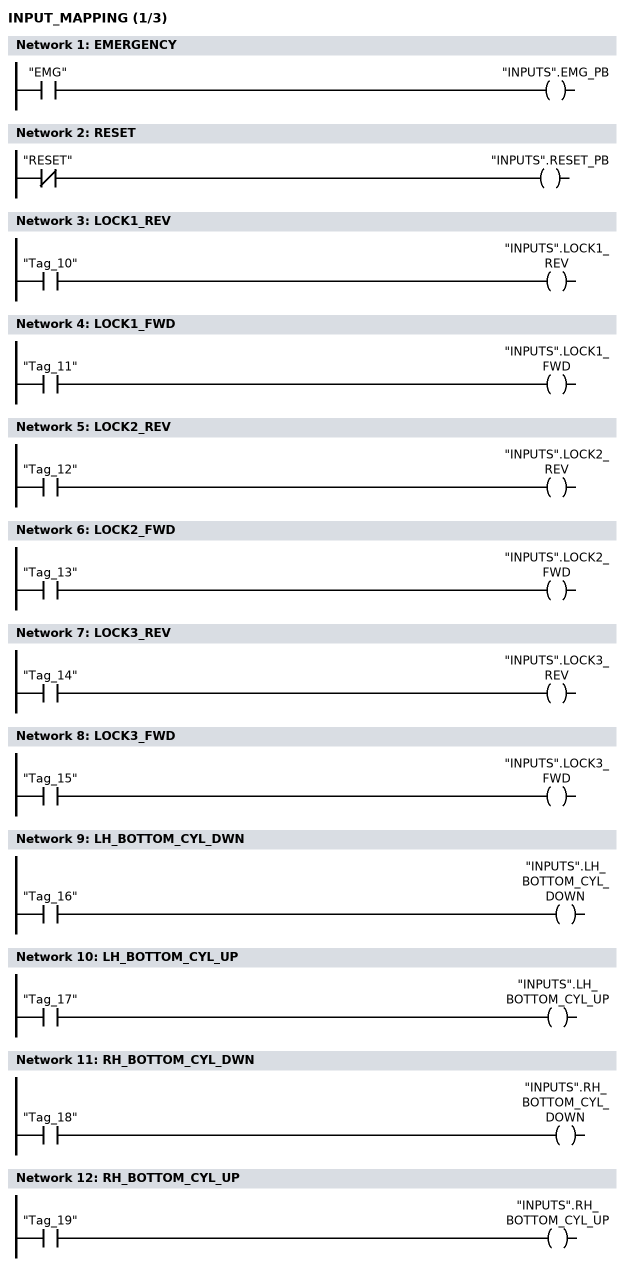
   RUNG wire#powerrail
      Contact( "EMG" )
      Coil( "INPUTS".EMG_PB )
   END_RUNG
   // the same network as SCL:
   "INPUTS".EMG_PB := "EMG";
END_REGION

REGION Network 2: RESET
   RUNG wire#powerrail
      I_Contact( "RESET" )
      Coil( "INPUTS".RESET_PB )
   END_RUNG
   // the same network as SCL:
   "INPUTS".RESET_PB := NOT "RESET";
END_REGION

REGION Network 3: LOCK1_REV
   RUNG wire#powerrail
      Contact( "Tag_10" )
      Coil( "INPUTS".LOCK1_REV )
   END_RUNG
   // the same network as SCL:
   "INPUTS".LOCK1_REV := "Tag_10";
END_REGION

REGION Network 4: LOCK1_FWD
   RUNG wire#powerrail
      Contact( "Tag_11" )
      Coil( "INPUTS".LOCK1_FWD )
   END_RUNG
   // the same network as SCL:
   "INPUTS".LOCK1_FWD := "Tag_11";
END_REGION

REGION Network 5: LOCK2_REV
   RUNG wire#powerrail
      Contact( "Tag_12" )
      Coil( "INPUTS".LOCK2_REV )
   END_RUNG
   // the same network as SCL:
   "INPUTS".LOCK2_REV := "Tag_12";
END_REGION

REGION Network 6: LOCK2_FWD
   RUNG wire#powerrail
      Contact( "Tag_13" )
      Coil( "INPUTS".LOCK2_FWD )
   END_RUNG
   // the same network as SCL:
   "INPUTS".LOCK2_FWD := "Tag_13";
END_REGION

REGION Network 7: LOCK3_REV
   RUNG wire#powerrail
      Contact( "Tag_14" )
      Coil( "INPUTS".LOCK3_REV )
   END_RUNG
   // the same network as SCL:
   "INPUTS".LOCK3_REV := "Tag_14";
END_REGION

REGION Network 8: LOCK3_FWD
   RUNG wire#powerrail
      Contact( "Tag_15" )
      Coil( "INPUTS".LOCK3_FWD )
   END_RUNG
   // the same network as SCL:
   "INPUTS".LOCK3_FWD := "Tag_15";
END_REGION

REGION Network 9: LH_BOTTOM_CYL_DWN
   RUNG wire#powerrail
      Contact( "Tag_16" )
      Coil( "INPUTS".LH_BOTTOM_CYL_DOWN )
   END_RUNG
   // the same network as SCL:
   "INPUTS".LH_BOTTOM_CYL_DOWN := "Tag_16";
END_REGION

REGION Network 10: LH_BOTTOM_CYL_UP
   RUNG wire#powerrail
      Contact( "Tag_17" )
      Coil( "INPUTS".LH_BOTTOM_CYL_UP )
   END_RUNG
   // the same network as SCL:
   "INPUTS".LH_BOTTOM_CYL_UP := "Tag_17";
END_REGION

REGION Network 11: RH_BOTTOM_CYL_DWN
   RUNG wire#powerrail
      Contact( "Tag_18" )
      Coil( "INPUTS".RH_BOTTOM_CYL_DOWN )
   END_RUNG
   // the same network as SCL:
   "INPUTS".RH_BOTTOM_CYL_DOWN := "Tag_18";
END_REGION

REGION Network 12: RH_BOTTOM_CYL_UP
   RUNG wire#powerrail
      Contact( "Tag_19" )
      Coil( "INPUTS".RH_BOTTOM_CYL_UP )
   END_RUNG
   // the same network as SCL:
   "INPUTS".RH_BOTTOM_CYL_UP := "Tag_19";
END_REGION

REGION Network 13: PUNCH_CYL1_REV
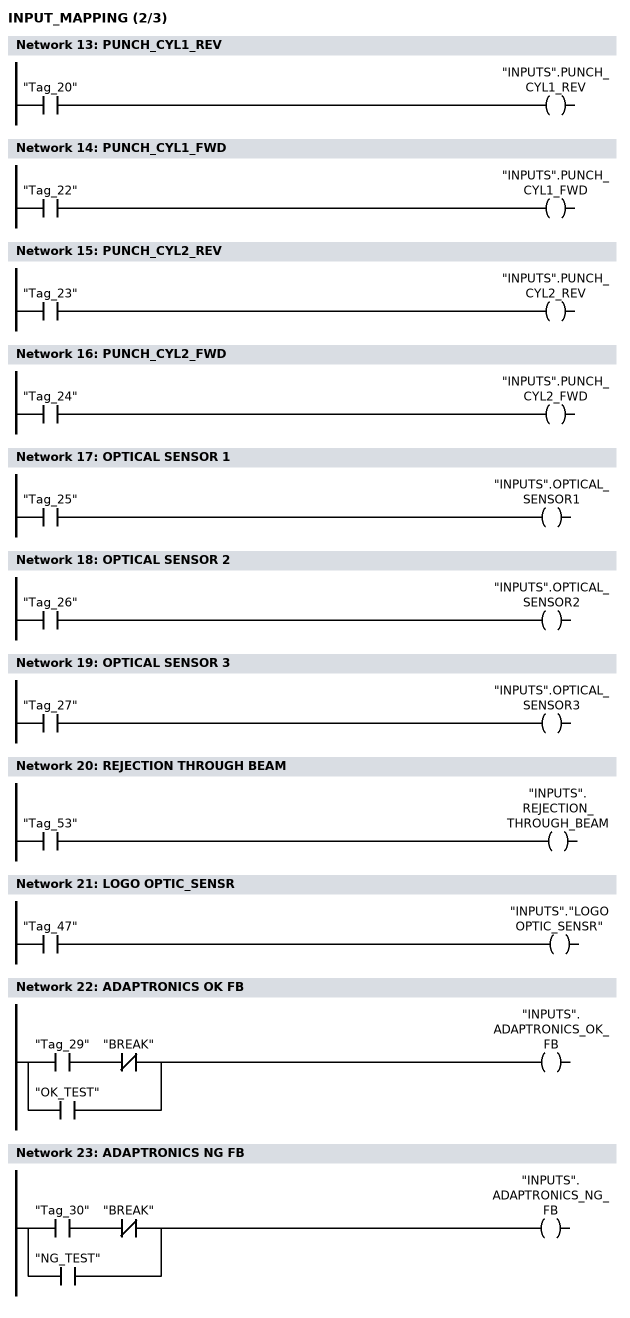
   RUNG wire#powerrail
      Contact( "Tag_20" )
      Coil( "INPUTS".PUNCH_CYL1_REV )
   END_RUNG
   // the same network as SCL:
   "INPUTS".PUNCH_CYL1_REV := "Tag_20";
END_REGION

REGION Network 14: PUNCH_CYL1_FWD
   RUNG wire#powerrail
      Contact( "Tag_22" )
      Coil( "INPUTS".PUNCH_CYL1_FWD )
   END_RUNG
   // the same network as SCL:
   "INPUTS".PUNCH_CYL1_FWD := "Tag_22";
END_REGION

REGION Network 15: PUNCH_CYL2_REV
   RUNG wire#powerrail
      Contact( "Tag_23" )
      Coil( "INPUTS".PUNCH_CYL2_REV )
   END_RUNG
   // the same network as SCL:
   "INPUTS".PUNCH_CYL2_REV := "Tag_23";
END_REGION

REGION Network 16: PUNCH_CYL2_FWD
   RUNG wire#powerrail
      Contact( "Tag_24" )
      Coil( "INPUTS".PUNCH_CYL2_FWD )
   END_RUNG
   // the same network as SCL:
   "INPUTS".PUNCH_CYL2_FWD := "Tag_24";
END_REGION

REGION Network 17: OPTICAL SENSOR 1
   RUNG wire#powerrail
      Contact( "Tag_25" )
      Coil( "INPUTS".OPTICAL_SENSOR1 )
   END_RUNG
   // the same network as SCL:
   "INPUTS".OPTICAL_SENSOR1 := "Tag_25";
END_REGION

REGION Network 18: OPTICAL SENSOR 2
   RUNG wire#powerrail
      Contact( "Tag_26" )
      Coil( "INPUTS".OPTICAL_SENSOR2 )
   END_RUNG
   // the same network as SCL:
   "INPUTS".OPTICAL_SENSOR2 := "Tag_26";
END_REGION

REGION Network 19: OPTICAL SENSOR 3
   RUNG wire#powerrail
      Contact( "Tag_27" )
      Coil( "INPUTS".OPTICAL_SENSOR3 )
   END_RUNG
   // the same network as SCL:
   "INPUTS".OPTICAL_SENSOR3 := "Tag_27";
END_REGION

REGION Network 20: REJECTION THROUGH BEAM
   RUNG wire#powerrail
      Contact( "Tag_53" )
      Coil( "INPUTS".REJECTION_THROUGH_BEAM )
   END_RUNG
   // the same network as SCL:
   "INPUTS".REJECTION_THROUGH_BEAM := "Tag_53";
END_REGION

REGION Network 21: LOGO OPTIC_SENSR
   RUNG wire#powerrail
      Contact( "Tag_47" )
      Coil( "INPUTS"."LOGO OPTIC_SENSR" )
   END_RUNG
   // the same network as SCL:
   "INPUTS"."LOGO OPTIC_SENSR" := "Tag_47";
END_REGION

REGION Network 22: ADAPTRONICS OK FB
   RUNG wire#powerrail
      Contact( "Tag_29" )
      I_Contact( "BREAK" )
      wire#w1
      Coil( "INPUTS".ADAPTRONICS_OK_FB )
   END_RUNG
   RUNG wire#powerrail
      Contact( "OK_TEST" )
   END_RUNG wire#w1
   // the same network as SCL:
   "INPUTS".ADAPTRONICS_OK_FB := ("Tag_29" AND NOT "BREAK") OR "OK_TEST";
END_REGION

REGION Network 23: ADAPTRONICS NG FB
   RUNG wire#powerrail
      Contact( "Tag_30" )
      I_Contact( "BREAK" )
      wire#w1
      Coil( "INPUTS".ADAPTRONICS_NG_FB )
   END_RUNG
   RUNG wire#powerrail
      Contact( "NG_TEST" )
   END_RUNG wire#w1
   // the same network as SCL:
   "INPUTS".ADAPTRONICS_NG_FB := ("Tag_30" AND NOT "BREAK") OR "NG_TEST";
END_REGION

REGION Network 24: ADAPTRONICS SEGMENT FB
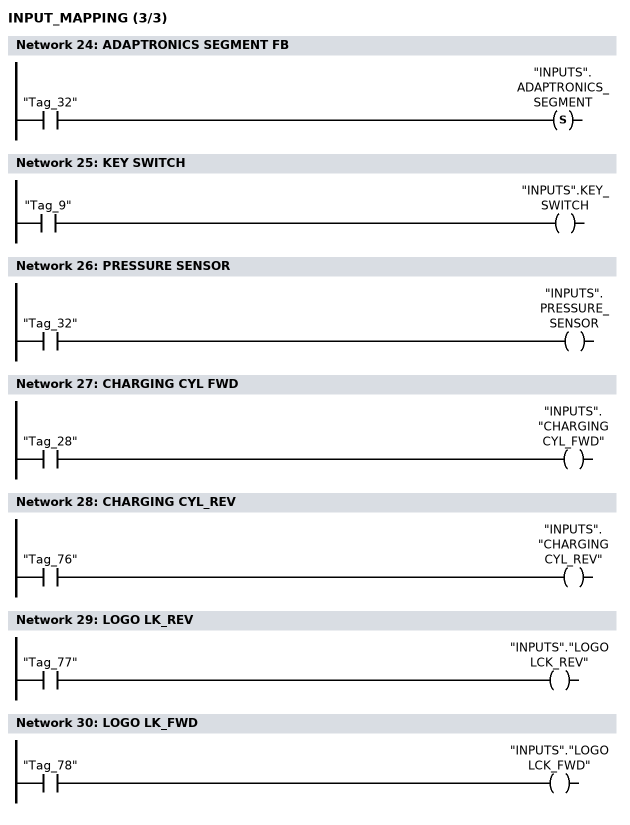
   RUNG wire#powerrail
      Contact( "Tag_32" )
      S_Coil( "INPUTS".ADAPTRONICS_SEGMENT )
   END_RUNG
   // the same network as SCL:
   IF "Tag_32" THEN "INPUTS".ADAPTRONICS_SEGMENT := TRUE; END_IF;
END_REGION

REGION Network 25: KEY SWITCH
   RUNG wire#powerrail
      Contact( "Tag_9" )
      Coil( "INPUTS".KEY_SWITCH )
   END_RUNG
   // the same network as SCL:
   "INPUTS".KEY_SWITCH := "Tag_9";
END_REGION

REGION Network 26: PRESSURE SENSOR
   RUNG wire#powerrail
      Contact( "Tag_32" )
      Coil( "INPUTS".PRESSURE_SENSOR )
   END_RUNG
   // the same network as SCL:
   "INPUTS".PRESSURE_SENSOR := "Tag_32";
END_REGION

REGION Network 27: CHARGING CYL FWD
   RUNG wire#powerrail
      Contact( "Tag_28" )
      Coil( "INPUTS"."CHARGING CYL_FWD" )
   END_RUNG
   // the same network as SCL:
   "INPUTS"."CHARGING CYL_FWD" := "Tag_28";
END_REGION

REGION Network 28: CHARGING CYL_REV
   RUNG wire#powerrail
      Contact( "Tag_76" )
      Coil( "INPUTS"."CHARGING CYL_REV" )
   END_RUNG
   // the same network as SCL:
   "INPUTS"."CHARGING CYL_REV" := "Tag_76";
END_REGION

REGION Network 29: LOGO LK_REV
   RUNG wire#powerrail
      Contact( "Tag_77" )
      Coil( "INPUTS"."LOGO LCK_REV" )
   END_RUNG
   // the same network as SCL:
   "INPUTS"."LOGO LCK_REV" := "Tag_77";
END_REGION

REGION Network 30: LOGO LK_FWD
   RUNG wire#powerrail
      Contact( "Tag_78" )
      Coil( "INPUTS"."LOGO LCK_FWD" )
   END_RUNG
   // the same network as SCL:
   "INPUTS"."LOGO LCK_FWD" := "Tag_78";
END_REGION
END_FUNCTION

FUNCTION "OUTPUT_MAPPING" : Void   // FC2, LAD
{ S7_Optimized_Access := 'TRUE' }
VERSION : 0.1
   VAR CONSTANT
      AMBER_ON : Bool;
   END_VAR
BEGIN

REGION Network 1: BUZZER
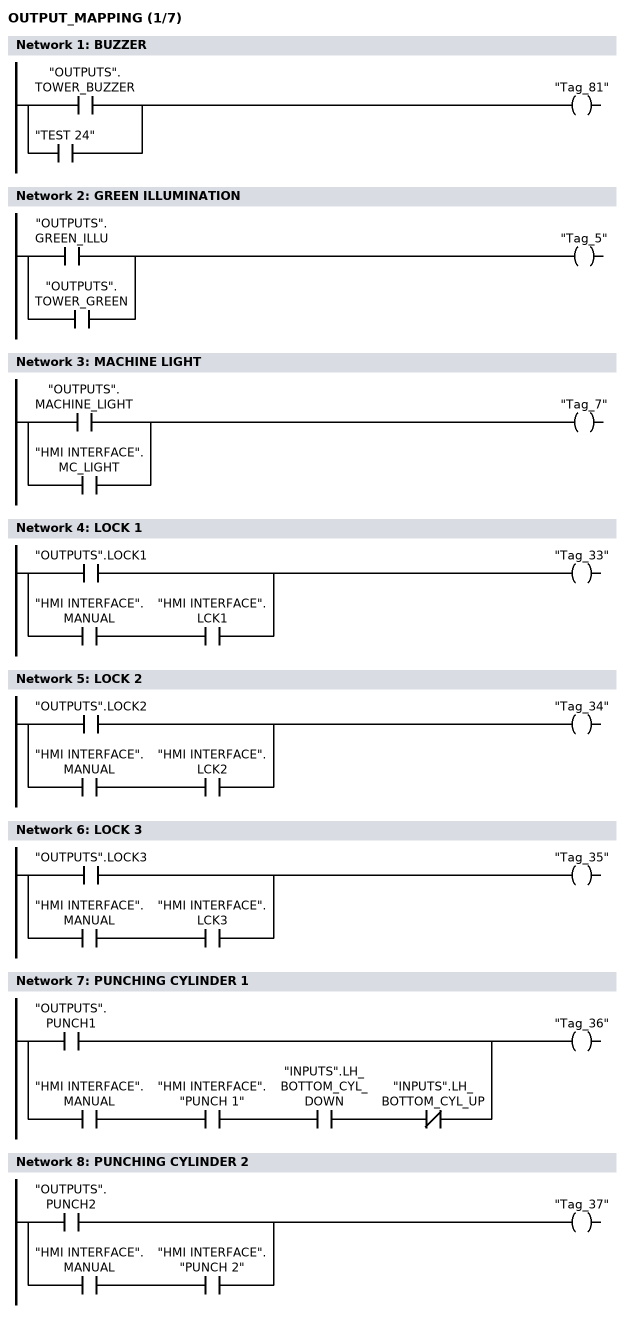
   RUNG wire#powerrail
      Contact( "OUTPUTS".TOWER_BUZZER )
      wire#w1
      Coil( "Tag_81" )
   END_RUNG
   RUNG wire#powerrail
      Contact( "TEST 24" )
   END_RUNG wire#w1
   // the same network as SCL:
   "Tag_81" := "OUTPUTS".TOWER_BUZZER OR "TEST 24";
END_REGION

REGION Network 2: GREEN ILLUMINATION
   RUNG wire#powerrail
      Contact( "OUTPUTS".GREEN_ILLU )
      wire#w1
      Coil( "Tag_5" )
   END_RUNG
   RUNG wire#powerrail
      Contact( "OUTPUTS".TOWER_GREEN )
   END_RUNG wire#w1
   // the same network as SCL:
   "Tag_5" := "OUTPUTS".GREEN_ILLU OR "OUTPUTS".TOWER_GREEN;
END_REGION

REGION Network 3: MACHINE LIGHT
   RUNG wire#powerrail
      Contact( "OUTPUTS".MACHINE_LIGHT )
      wire#w1
      Coil( "Tag_7" )
   END_RUNG
   RUNG wire#powerrail
      Contact( "HMI INTERFACE".MC_LIGHT )
   END_RUNG wire#w1
   // the same network as SCL:
   "Tag_7" := "OUTPUTS".MACHINE_LIGHT OR "HMI INTERFACE".MC_LIGHT;
END_REGION

REGION Network 4: LOCK 1
   RUNG wire#powerrail
      Contact( "OUTPUTS".LOCK1 )
      wire#w1
      Coil( "Tag_33" )
   END_RUNG
   RUNG wire#powerrail
      Contact( "HMI INTERFACE".MANUAL )
      Contact( "HMI INTERFACE".LCK1 )
   END_RUNG wire#w1
   // the same network as SCL:
   "Tag_33" := "OUTPUTS".LOCK1 OR ("HMI INTERFACE".MANUAL AND "HMI INTERFACE".LCK1);
END_REGION

REGION Network 5: LOCK 2
   RUNG wire#powerrail
      Contact( "OUTPUTS".LOCK2 )
      wire#w1
      Coil( "Tag_34" )
   END_RUNG
   RUNG wire#powerrail
      Contact( "HMI INTERFACE".MANUAL )
      Contact( "HMI INTERFACE".LCK2 )
   END_RUNG wire#w1
   // the same network as SCL:
   "Tag_34" := "OUTPUTS".LOCK2 OR ("HMI INTERFACE".MANUAL AND "HMI INTERFACE".LCK2);
END_REGION

REGION Network 6: LOCK 3
   RUNG wire#powerrail
      Contact( "OUTPUTS".LOCK3 )
      wire#w1
      Coil( "Tag_35" )
   END_RUNG
   RUNG wire#powerrail
      Contact( "HMI INTERFACE".MANUAL )
      Contact( "HMI INTERFACE".LCK3 )
   END_RUNG wire#w1
   // the same network as SCL:
   "Tag_35" := "OUTPUTS".LOCK3 OR ("HMI INTERFACE".MANUAL AND "HMI INTERFACE".LCK3);
END_REGION

REGION Network 7: PUNCHING CYLINDER 1
   RUNG wire#powerrail
      Contact( "OUTPUTS".PUNCH1 )
      wire#w1
      Coil( "Tag_36" )
   END_RUNG
   RUNG wire#powerrail
      Contact( "HMI INTERFACE".MANUAL )
      Contact( "HMI INTERFACE"."PUNCH 1" )
      Contact( "INPUTS".LH_BOTTOM_CYL_DOWN )
      I_Contact( "INPUTS".LH_BOTTOM_CYL_UP )
   END_RUNG wire#w1
   // the same network as SCL:
   "Tag_36" := "OUTPUTS".PUNCH1 OR ("HMI INTERFACE".MANUAL AND "HMI INTERFACE"."PUNCH 1" AND "INPUTS".LH_BOTTOM_CYL_DOWN AND NOT "INPUTS".LH_BOTTOM_CYL_UP);
END_REGION

REGION Network 8: PUNCHING CYLINDER 2
   RUNG wire#powerrail
      Contact( "OUTPUTS".PUNCH2 )
      wire#w1
      Coil( "Tag_37" )
   END_RUNG
   RUNG wire#powerrail
      Contact( "HMI INTERFACE".MANUAL )
      Contact( "HMI INTERFACE"."PUNCH 2" )
   END_RUNG wire#w1
   // the same network as SCL:
   "Tag_37" := "OUTPUTS".PUNCH2 OR ("HMI INTERFACE".MANUAL AND "HMI INTERFACE"."PUNCH 2");
END_REGION

REGION Network 9: LH_BOTTOM_CYL
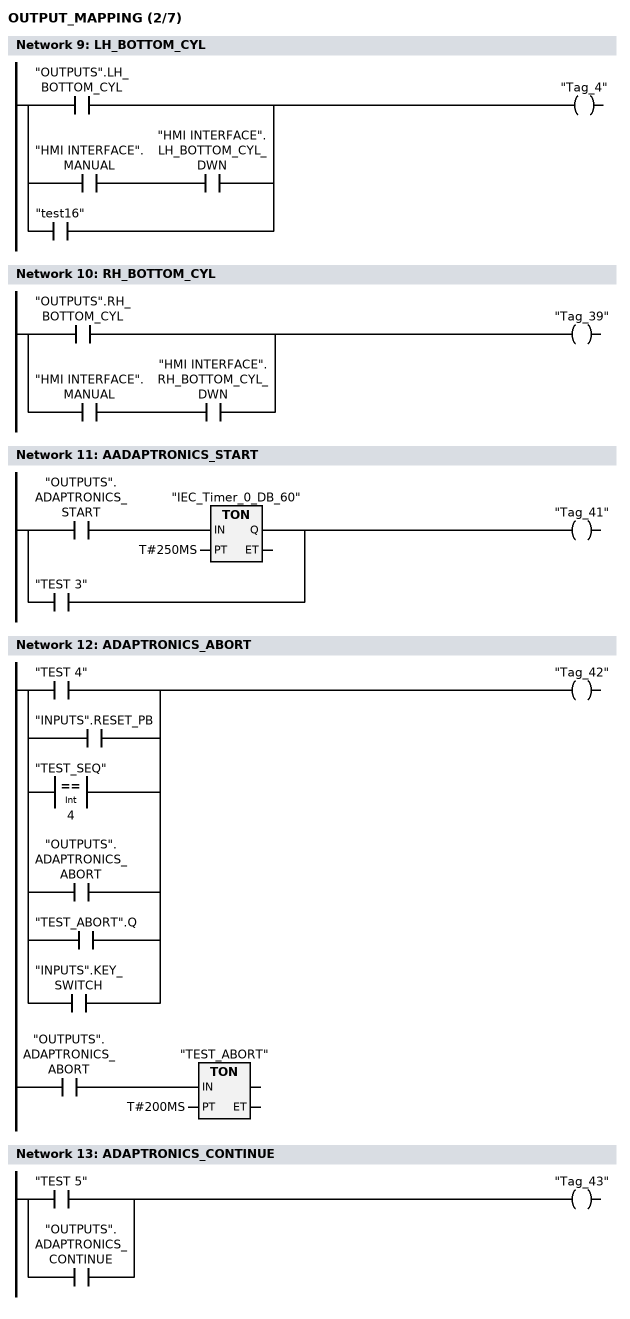
   RUNG wire#powerrail
      Contact( "OUTPUTS".LH_BOTTOM_CYL )
      wire#w1
      Coil( "Tag_4" )
   END_RUNG
   RUNG wire#powerrail
      Contact( "HMI INTERFACE".MANUAL )
      Contact( "HMI INTERFACE".LH_BOTTOM_CYL_DWN )
   END_RUNG wire#w1
   RUNG wire#powerrail
      Contact( "test16" )
   END_RUNG wire#w1
   // the same network as SCL:
   "Tag_4" := "OUTPUTS".LH_BOTTOM_CYL OR ("HMI INTERFACE".MANUAL AND "HMI INTERFACE".LH_BOTTOM_CYL_DWN) OR "test16";
END_REGION

REGION Network 10: RH_BOTTOM_CYL
   RUNG wire#powerrail
      Contact( "OUTPUTS".RH_BOTTOM_CYL )
      wire#w1
      Coil( "Tag_39" )
   END_RUNG
   RUNG wire#powerrail
      Contact( "HMI INTERFACE".MANUAL )
      Contact( "HMI INTERFACE".RH_BOTTOM_CYL_DWN )
   END_RUNG wire#w1
   // the same network as SCL:
   "Tag_39" := "OUTPUTS".RH_BOTTOM_CYL OR ("HMI INTERFACE".MANUAL AND "HMI INTERFACE".RH_BOTTOM_CYL_DWN);
END_REGION

REGION Network 11: AADAPTRONICS_START
   "IEC_Timer_0_DB_60".TON(IN := "OUTPUTS".ADAPTRONICS_START, PT := T#250MS);
   "Tag_41" := "IEC_Timer_0_DB_60".Q OR "TEST 3";
END_REGION

REGION Network 12: ADAPTRONICS_ABORT
   "Tag_42" := "TEST 4" OR "INPUTS".RESET_PB OR ("TEST_SEQ" = 4) OR "OUTPUTS".ADAPTRONICS_ABORT OR "TEST_ABORT".Q OR "INPUTS".KEY_SWITCH;
   "TEST_ABORT".TON(IN := "OUTPUTS".ADAPTRONICS_ABORT, PT := T#200MS);
END_REGION

REGION Network 13: ADAPTRONICS_CONTINUE
   RUNG wire#powerrail
      Contact( "TEST 5" )
      wire#w1
      Coil( "Tag_43" )
   END_RUNG
   RUNG wire#powerrail
      Contact( "OUTPUTS".ADAPTRONICS_CONTINUE )
   END_RUNG wire#w1
   // the same network as SCL:
   "Tag_43" := "TEST 5" OR "OUTPUTS".ADAPTRONICS_CONTINUE;
END_REGION

REGION Network 14: RELAY 1 / RED
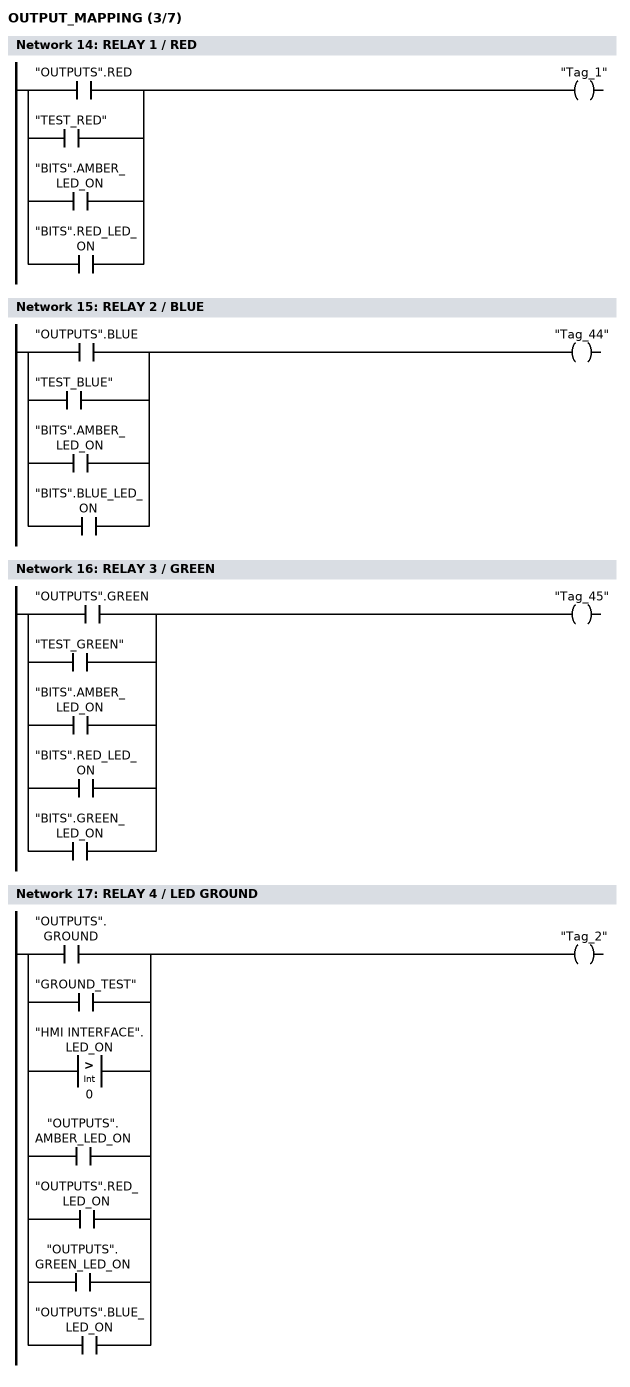
   RUNG wire#powerrail
      Contact( "OUTPUTS".RED )
      wire#w1
      Coil( "Tag_1" )
   END_RUNG
   RUNG wire#powerrail
      Contact( "TEST_RED" )
   END_RUNG wire#w1
   RUNG wire#powerrail
      Contact( "BITS".AMBER_LED_ON )
   END_RUNG wire#w1
   RUNG wire#powerrail
      Contact( "BITS".RED_LED_ON )
   END_RUNG wire#w1
   // the same network as SCL:
   "Tag_1" := "OUTPUTS".RED OR "TEST_RED" OR "BITS".AMBER_LED_ON OR "BITS".RED_LED_ON;
END_REGION

REGION Network 15: RELAY 2 / BLUE
   RUNG wire#powerrail
      Contact( "OUTPUTS".BLUE )
      wire#w1
      Coil( "Tag_44" )
   END_RUNG
   RUNG wire#powerrail
      Contact( "TEST_BLUE" )
   END_RUNG wire#w1
   RUNG wire#powerrail
      Contact( "BITS".AMBER_LED_ON )
   END_RUNG wire#w1
   RUNG wire#powerrail
      Contact( "BITS".BLUE_LED_ON )
   END_RUNG wire#w1
   // the same network as SCL:
   "Tag_44" := "OUTPUTS".BLUE OR "TEST_BLUE" OR "BITS".AMBER_LED_ON OR "BITS".BLUE_LED_ON;
END_REGION

REGION Network 16: RELAY 3 / GREEN
   RUNG wire#powerrail
      Contact( "OUTPUTS".GREEN )
      wire#w1
      Coil( "Tag_45" )
   END_RUNG
   RUNG wire#powerrail
      Contact( "TEST_GREEN" )
   END_RUNG wire#w1
   RUNG wire#powerrail
      Contact( "BITS".AMBER_LED_ON )
   END_RUNG wire#w1
   RUNG wire#powerrail
      Contact( "BITS".RED_LED_ON )
   END_RUNG wire#w1
   RUNG wire#powerrail
      Contact( "BITS".GREEN_LED_ON )
   END_RUNG wire#w1
   // the same network as SCL:
   "Tag_45" := "OUTPUTS".GREEN OR "TEST_GREEN" OR "BITS".AMBER_LED_ON OR "BITS".RED_LED_ON OR "BITS".GREEN_LED_ON;
END_REGION

REGION Network 17: RELAY 4 / LED GROUND
   RUNG wire#powerrail
      Contact( "OUTPUTS".GROUND )
      wire#w1
      Coil( "Tag_2" )
   END_RUNG
   RUNG wire#powerrail
      Contact( "GROUND_TEST" )
   END_RUNG wire#w1
   RUNG wire#powerrail
      { S7_Templates := "SrcType := Int" } GT_Contact(in1 := "HMI INTERFACE".LED_ON, in2 := 0)
   END_RUNG wire#w1
   RUNG wire#powerrail
      Contact( "OUTPUTS".AMBER_LED_ON )
   END_RUNG wire#w1
   RUNG wire#powerrail
      Contact( "OUTPUTS".RED_LED_ON )
   END_RUNG wire#w1
   RUNG wire#powerrail
      Contact( "OUTPUTS".GREEN_LED_ON )
   END_RUNG wire#w1
   RUNG wire#powerrail
      Contact( "OUTPUTS".BLUE_LED_ON )
   END_RUNG wire#w1
   // the same network as SCL:
   "Tag_2" := "OUTPUTS".GROUND OR "GROUND_TEST" OR ("HMI INTERFACE".LED_ON > 0) OR "OUTPUTS".AMBER_LED_ON OR "OUTPUTS".RED_LED_ON OR "OUTPUTS".GREEN_LED_ON OR "OUTPUTS".BLUE_LED_ON;
END_REGION

REGION Network 18: X1
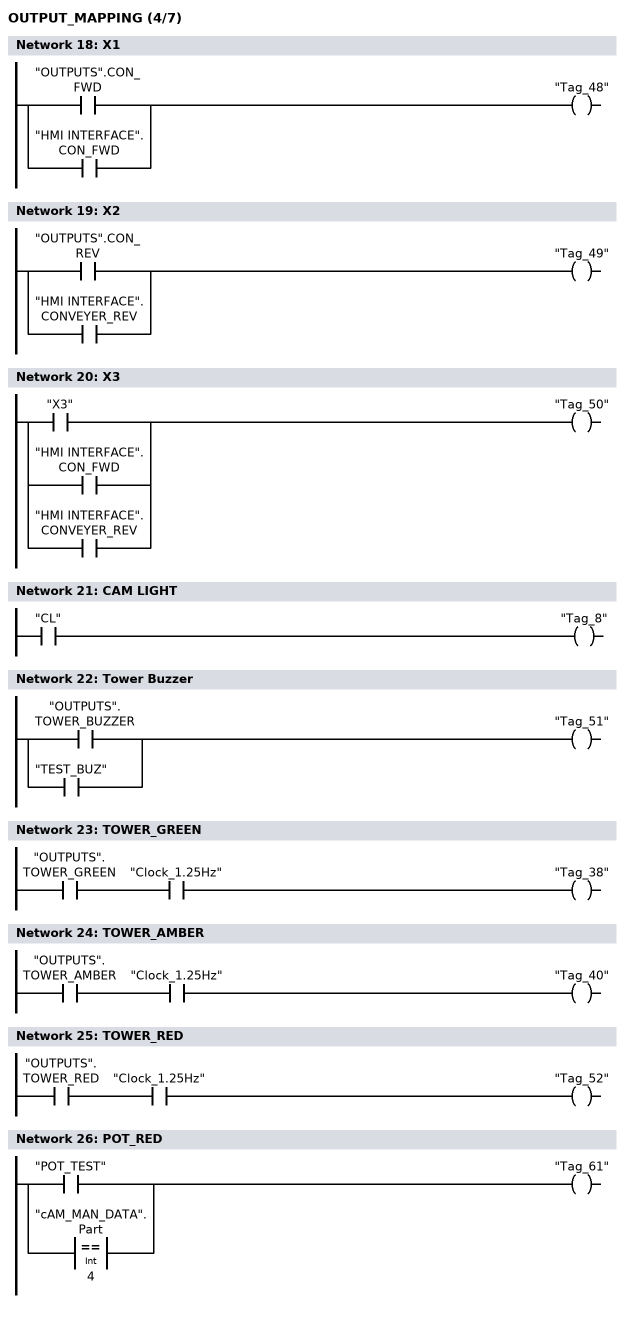
   RUNG wire#powerrail
      Contact( "OUTPUTS".CON_FWD )
      wire#w1
      Coil( "Tag_48" )
   END_RUNG
   RUNG wire#powerrail
      Contact( "HMI INTERFACE".CON_FWD )
   END_RUNG wire#w1
   // the same network as SCL:
   "Tag_48" := "OUTPUTS".CON_FWD OR "HMI INTERFACE".CON_FWD;
END_REGION

REGION Network 19: X2
   RUNG wire#powerrail
      Contact( "OUTPUTS".CON_REV )
      wire#w1
      Coil( "Tag_49" )
   END_RUNG
   RUNG wire#powerrail
      Contact( "HMI INTERFACE".CONVEYER_REV )
   END_RUNG wire#w1
   // the same network as SCL:
   "Tag_49" := "OUTPUTS".CON_REV OR "HMI INTERFACE".CONVEYER_REV;
END_REGION

REGION Network 20: X3
   RUNG wire#powerrail
      Contact( "X3" )
      wire#w1
      Coil( "Tag_50" )
   END_RUNG
   RUNG wire#powerrail
      Contact( "HMI INTERFACE".CON_FWD )
   END_RUNG wire#w1
   RUNG wire#powerrail
      Contact( "HMI INTERFACE".CONVEYER_REV )
   END_RUNG wire#w1
   // the same network as SCL:
   "Tag_50" := "X3" OR "HMI INTERFACE".CON_FWD OR "HMI INTERFACE".CONVEYER_REV;
END_REGION

REGION Network 21: CAM LIGHT
   RUNG wire#powerrail
      Contact( "CL" )
      Coil( "Tag_8" )
   END_RUNG
   // the same network as SCL:
   "Tag_8" := "CL";
END_REGION

REGION Network 22: Tower Buzzer
   RUNG wire#powerrail
      Contact( "OUTPUTS".TOWER_BUZZER )
      wire#w1
      Coil( "Tag_51" )
   END_RUNG
   RUNG wire#powerrail
      Contact( "TEST_BUZ" )
   END_RUNG wire#w1
   // the same network as SCL:
   "Tag_51" := "OUTPUTS".TOWER_BUZZER OR "TEST_BUZ";
END_REGION

REGION Network 23: TOWER_GREEN
   RUNG wire#powerrail
      Contact( "OUTPUTS".TOWER_GREEN )
      Contact( "Clock_1.25Hz" )
      Coil( "Tag_38" )
   END_RUNG
   // the same network as SCL:
   "Tag_38" := "OUTPUTS".TOWER_GREEN AND "Clock_1.25Hz";
END_REGION

REGION Network 24: TOWER_AMBER
   RUNG wire#powerrail
      Contact( "OUTPUTS".TOWER_AMBER )
      Contact( "Clock_1.25Hz" )
      Coil( "Tag_40" )
   END_RUNG
   // the same network as SCL:
   "Tag_40" := "OUTPUTS".TOWER_AMBER AND "Clock_1.25Hz";
END_REGION

REGION Network 25: TOWER_RED
   RUNG wire#powerrail
      Contact( "OUTPUTS".TOWER_RED )
      Contact( "Clock_1.25Hz" )
      Coil( "Tag_52" )
   END_RUNG
   // the same network as SCL:
   "Tag_52" := "OUTPUTS".TOWER_RED AND "Clock_1.25Hz";
END_REGION

REGION Network 26: POT_RED
   RUNG wire#powerrail
      Contact( "POT_TEST" )
      wire#w1
      Coil( "Tag_61" )
   END_RUNG
   RUNG wire#powerrail
      { S7_Templates := "SrcType := Int" } EQ_Contact(in1 := "cAM_MAN_DATA".Part, in2 := 4)
   END_RUNG wire#w1
   // the same network as SCL:
   "Tag_61" := "POT_TEST" OR ("cAM_MAN_DATA".Part = 4);
END_REGION

REGION Network 27: RELAY BLUE
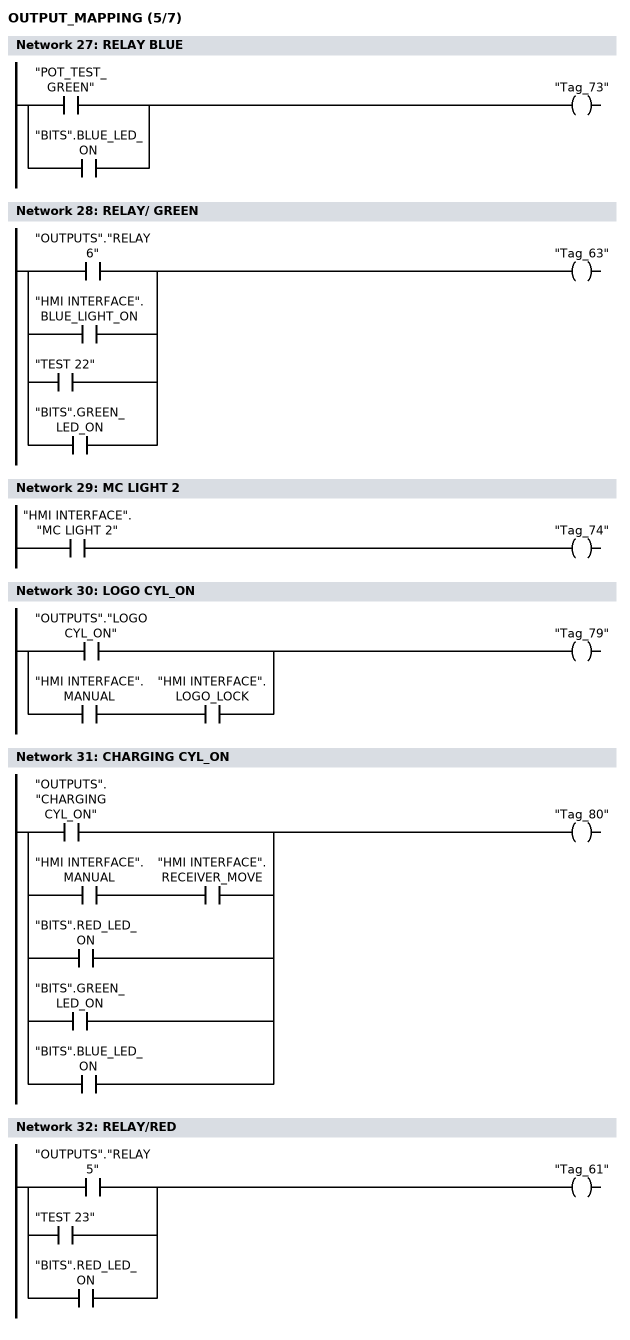
   RUNG wire#powerrail
      Contact( "POT_TEST_GREEN" )
      wire#w1
      Coil( "Tag_73" )
   END_RUNG
   RUNG wire#powerrail
      Contact( "BITS".BLUE_LED_ON )
   END_RUNG wire#w1
   // the same network as SCL:
   "Tag_73" := "POT_TEST_GREEN" OR "BITS".BLUE_LED_ON;
END_REGION

REGION Network 28: RELAY/ GREEN
   RUNG wire#powerrail
      Contact( "OUTPUTS"."RELAY 6" )
      wire#w1
      Coil( "Tag_63" )
   END_RUNG
   RUNG wire#powerrail
      Contact( "HMI INTERFACE".BLUE_LIGHT_ON )
   END_RUNG wire#w1
   RUNG wire#powerrail
      Contact( "TEST 22" )
   END_RUNG wire#w1
   RUNG wire#powerrail
      Contact( "BITS".GREEN_LED_ON )
   END_RUNG wire#w1
   // the same network as SCL:
   "Tag_63" := "OUTPUTS"."RELAY 6" OR "HMI INTERFACE".BLUE_LIGHT_ON OR "TEST 22" OR "BITS".GREEN_LED_ON;
END_REGION

REGION Network 29: MC LIGHT 2
   RUNG wire#powerrail
      Contact( "HMI INTERFACE"."MC LIGHT 2" )
      Coil( "Tag_74" )
   END_RUNG
   // the same network as SCL:
   "Tag_74" := "HMI INTERFACE"."MC LIGHT 2";
END_REGION

REGION Network 30: LOGO CYL_ON
   RUNG wire#powerrail
      Contact( "OUTPUTS"."LOGO CYL_ON" )
      wire#w1
      Coil( "Tag_79" )
   END_RUNG
   RUNG wire#powerrail
      Contact( "HMI INTERFACE".MANUAL )
      Contact( "HMI INTERFACE".LOGO_LOCK )
   END_RUNG wire#w1
   // the same network as SCL:
   "Tag_79" := "OUTPUTS"."LOGO CYL_ON" OR ("HMI INTERFACE".MANUAL AND "HMI INTERFACE".LOGO_LOCK);
END_REGION

REGION Network 31: CHARGING CYL_ON
   RUNG wire#powerrail
      Contact( "OUTPUTS"."CHARGING CYL_ON" )
      wire#w1
      Coil( "Tag_80" )
   END_RUNG
   RUNG wire#powerrail
      Contact( "HMI INTERFACE".MANUAL )
      Contact( "HMI INTERFACE".RECEIVER_MOVE )
   END_RUNG wire#w1
   RUNG wire#powerrail
      Contact( "BITS".RED_LED_ON )
   END_RUNG wire#w1
   RUNG wire#powerrail
      Contact( "BITS".GREEN_LED_ON )
   END_RUNG wire#w1
   RUNG wire#powerrail
      Contact( "BITS".BLUE_LED_ON )
   END_RUNG wire#w1
   // the same network as SCL:
   "Tag_80" := "OUTPUTS"."CHARGING CYL_ON" OR ("HMI INTERFACE".MANUAL AND "HMI INTERFACE".RECEIVER_MOVE) OR "BITS".RED_LED_ON OR "BITS".GREEN_LED_ON OR "BITS".BLUE_LED_ON;
END_REGION

REGION Network 32: RELAY/RED
   RUNG wire#powerrail
      Contact( "OUTPUTS"."RELAY 5" )
      wire#w1
      Coil( "Tag_61" )
   END_RUNG
   RUNG wire#powerrail
      Contact( "TEST 23" )
   END_RUNG wire#w1
   RUNG wire#powerrail
      Contact( "BITS".RED_LED_ON )
   END_RUNG wire#w1
   // the same network as SCL:
   "Tag_61" := "OUTPUTS"."RELAY 5" OR "TEST 23" OR "BITS".RED_LED_ON;
END_REGION

REGION Network 33: AMBER / RED COMMON
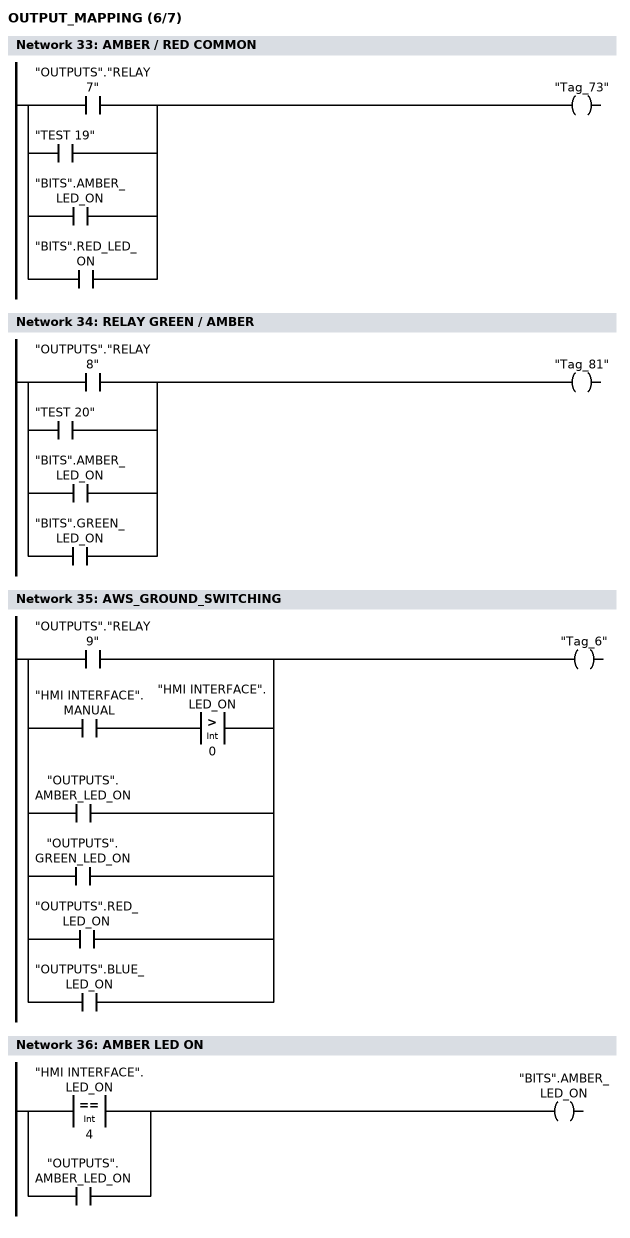
   RUNG wire#powerrail
      Contact( "OUTPUTS"."RELAY 7" )
      wire#w1
      Coil( "Tag_73" )
   END_RUNG
   RUNG wire#powerrail
      Contact( "TEST 19" )
   END_RUNG wire#w1
   RUNG wire#powerrail
      Contact( "BITS".AMBER_LED_ON )
   END_RUNG wire#w1
   RUNG wire#powerrail
      Contact( "BITS".RED_LED_ON )
   END_RUNG wire#w1
   // the same network as SCL:
   "Tag_73" := "OUTPUTS"."RELAY 7" OR "TEST 19" OR "BITS".AMBER_LED_ON OR "BITS".RED_LED_ON;
END_REGION

REGION Network 34: RELAY GREEN / AMBER
   RUNG wire#powerrail
      Contact( "OUTPUTS"."RELAY 8" )
      wire#w1
      Coil( "Tag_81" )
   END_RUNG
   RUNG wire#powerrail
      Contact( "TEST 20" )
   END_RUNG wire#w1
   RUNG wire#powerrail
      Contact( "BITS".AMBER_LED_ON )
   END_RUNG wire#w1
   RUNG wire#powerrail
      Contact( "BITS".GREEN_LED_ON )
   END_RUNG wire#w1
   // the same network as SCL:
   "Tag_81" := "OUTPUTS"."RELAY 8" OR "TEST 20" OR "BITS".AMBER_LED_ON OR "BITS".GREEN_LED_ON;
END_REGION

REGION Network 35: AWS_GROUND_SWITCHING
   RUNG wire#powerrail
      Contact( "OUTPUTS"."RELAY 9" )
      wire#w1
      Coil( "Tag_6" )
   END_RUNG
   RUNG wire#powerrail
      Contact( "HMI INTERFACE".MANUAL )
      { S7_Templates := "SrcType := Int" } GT_Contact(in1 := "HMI INTERFACE".LED_ON, in2 := 0)
   END_RUNG wire#w1
   RUNG wire#powerrail
      Contact( "OUTPUTS".AMBER_LED_ON )
   END_RUNG wire#w1
   RUNG wire#powerrail
      Contact( "OUTPUTS".GREEN_LED_ON )
   END_RUNG wire#w1
   RUNG wire#powerrail
      Contact( "OUTPUTS".RED_LED_ON )
   END_RUNG wire#w1
   RUNG wire#powerrail
      Contact( "OUTPUTS".BLUE_LED_ON )
   END_RUNG wire#w1
   // the same network as SCL:
   "Tag_6" := "OUTPUTS"."RELAY 9" OR ("HMI INTERFACE".MANUAL AND ("HMI INTERFACE".LED_ON > 0)) OR "OUTPUTS".AMBER_LED_ON OR "OUTPUTS".GREEN_LED_ON OR "OUTPUTS".RED_LED_ON OR "OUTPUTS".BLUE_LED_ON;
END_REGION

REGION Network 36: AMBER LED ON
   RUNG wire#powerrail
      { S7_Templates := "SrcType := Int" } EQ_Contact(in1 := "HMI INTERFACE".LED_ON, in2 := 4)
      wire#w1
      Coil( "BITS".AMBER_LED_ON )
   END_RUNG
   RUNG wire#powerrail
      Contact( "OUTPUTS".AMBER_LED_ON )
   END_RUNG wire#w1
   // the same network as SCL:
   "BITS".AMBER_LED_ON := ("HMI INTERFACE".LED_ON = 4) OR "OUTPUTS".AMBER_LED_ON;
END_REGION

REGION Network 37: RED_LED_ON
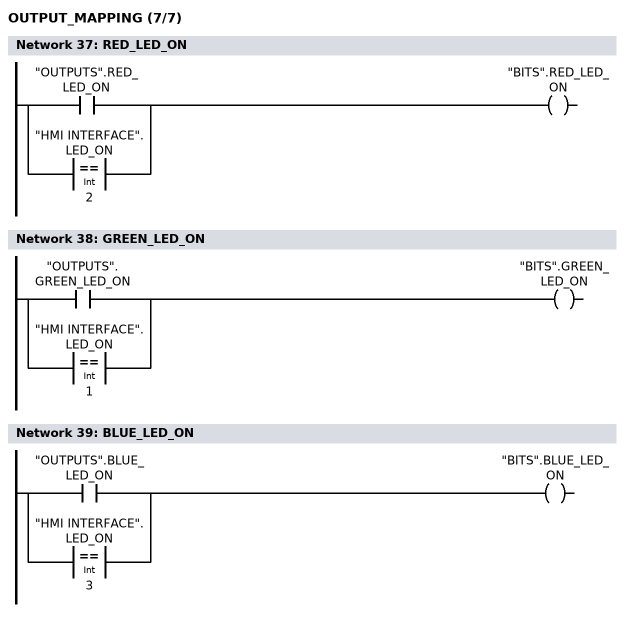
   RUNG wire#powerrail
      Contact( "OUTPUTS".RED_LED_ON )
      wire#w1
      Coil( "BITS".RED_LED_ON )
   END_RUNG
   RUNG wire#powerrail
      { S7_Templates := "SrcType := Int" } EQ_Contact(in1 := "HMI INTERFACE".LED_ON, in2 := 2)
   END_RUNG wire#w1
   // the same network as SCL:
   "BITS".RED_LED_ON := "OUTPUTS".RED_LED_ON OR ("HMI INTERFACE".LED_ON = 2);
END_REGION

REGION Network 38: GREEN_LED_ON
   RUNG wire#powerrail
      Contact( "OUTPUTS".GREEN_LED_ON )
      wire#w1
      Coil( "BITS".GREEN_LED_ON )
   END_RUNG
   RUNG wire#powerrail
      { S7_Templates := "SrcType := Int" } EQ_Contact(in1 := "HMI INTERFACE".LED_ON, in2 := 1)
   END_RUNG wire#w1
   // the same network as SCL:
   "BITS".GREEN_LED_ON := "OUTPUTS".GREEN_LED_ON OR ("HMI INTERFACE".LED_ON = 1);
END_REGION

REGION Network 39: BLUE_LED_ON
   RUNG wire#powerrail
      Contact( "OUTPUTS".BLUE_LED_ON )
      wire#w1
      Coil( "BITS".BLUE_LED_ON )
   END_RUNG
   RUNG wire#powerrail
      { S7_Templates := "SrcType := Int" } EQ_Contact(in1 := "HMI INTERFACE".LED_ON, in2 := 3)
   END_RUNG wire#w1
   // the same network as SCL:
   "BITS".BLUE_LED_ON := "OUTPUTS".BLUE_LED_ON OR ("HMI INTERFACE".LED_ON = 3);
END_REGION
END_FUNCTION

FUNCTION "ERROR_MESSAGES" : Void   // FC4, LAD
{ S7_Optimized_Access := 'TRUE' }
VERSION : 0.1
   VAR_TEMP
      ERROR_BIT1 : Bool;
   END_VAR
BEGIN

REGION Network 1: LOCK1_FWD_REED_MISSING
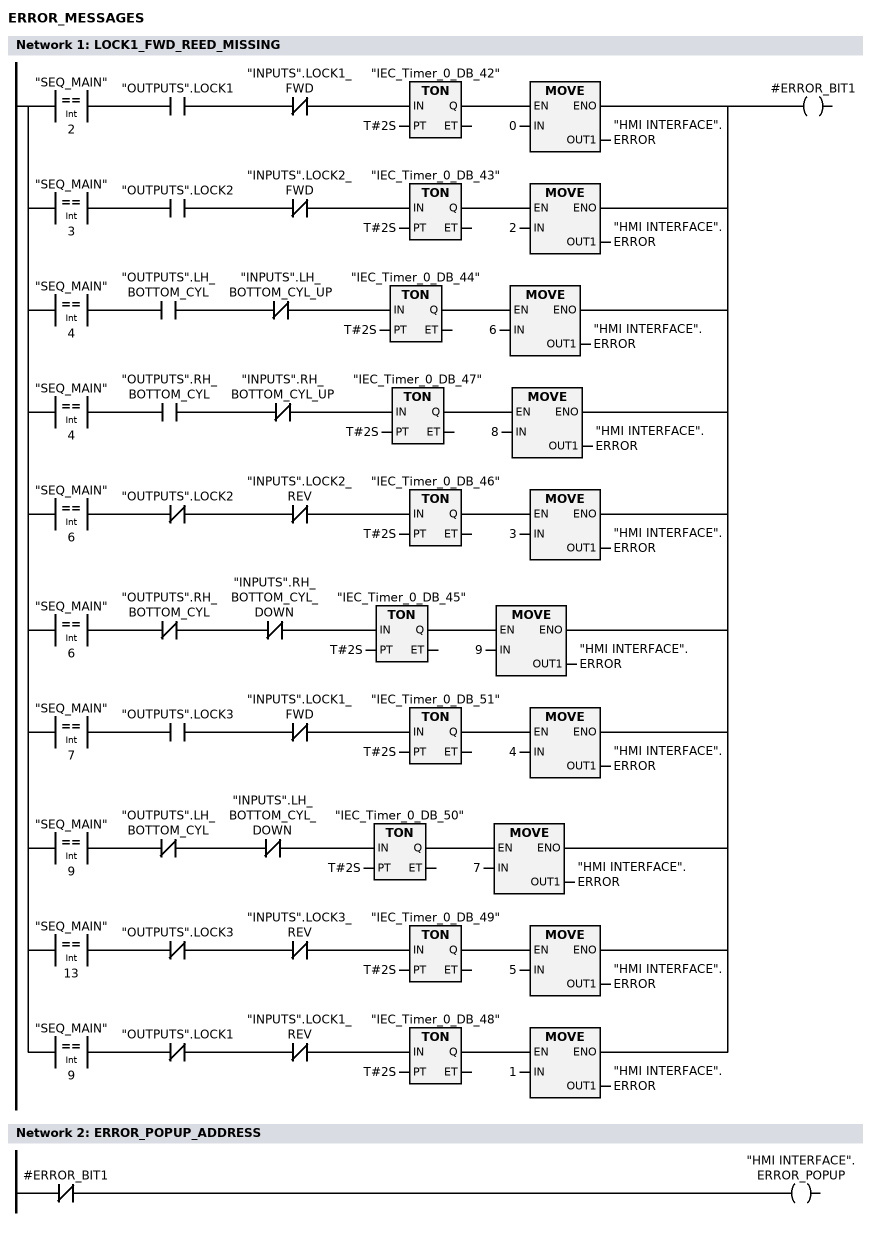
   "IEC_Timer_0_DB_42".TON(IN := ("SEQ_MAIN" = 2) AND "OUTPUTS".LOCK1 AND NOT "INPUTS".LOCK1_FWD, PT := T#2S);
   IF "IEC_Timer_0_DB_42".Q THEN "HMI INTERFACE".ERROR := 0; END_IF;
   "IEC_Timer_0_DB_43".TON(IN := ("SEQ_MAIN" = 3) AND "OUTPUTS".LOCK2 AND NOT "INPUTS".LOCK2_FWD, PT := T#2S);
   IF "IEC_Timer_0_DB_43".Q THEN "HMI INTERFACE".ERROR := 2; END_IF;
   "IEC_Timer_0_DB_44".TON(IN := ("SEQ_MAIN" = 4) AND "OUTPUTS".LH_BOTTOM_CYL AND NOT "INPUTS".LH_BOTTOM_CYL_UP,
                           PT := T#2S);
   IF "IEC_Timer_0_DB_44".Q THEN "HMI INTERFACE".ERROR := 6; END_IF;
   "IEC_Timer_0_DB_47".TON(IN := ("SEQ_MAIN" = 4) AND "OUTPUTS".RH_BOTTOM_CYL AND NOT "INPUTS".RH_BOTTOM_CYL_UP,
                           PT := T#2S);
   IF "IEC_Timer_0_DB_47".Q THEN "HMI INTERFACE".ERROR := 8; END_IF;
   "IEC_Timer_0_DB_46".TON(IN := ("SEQ_MAIN" = 6) AND NOT "OUTPUTS".LOCK2 AND NOT "INPUTS".LOCK2_REV,
                           PT := T#2S);
   IF "IEC_Timer_0_DB_46".Q THEN "HMI INTERFACE".ERROR := 3; END_IF;
   "IEC_Timer_0_DB_45".TON(IN := ("SEQ_MAIN" = 6) AND NOT "OUTPUTS".RH_BOTTOM_CYL AND NOT "INPUTS".RH_BOTTOM_CYL_DOWN,
                           PT := T#2S);
   IF "IEC_Timer_0_DB_45".Q THEN "HMI INTERFACE".ERROR := 9; END_IF;
   "IEC_Timer_0_DB_51".TON(IN := ("SEQ_MAIN" = 7) AND "OUTPUTS".LOCK3 AND NOT "INPUTS".LOCK1_FWD, PT := T#2S);
   IF "IEC_Timer_0_DB_51".Q THEN "HMI INTERFACE".ERROR := 4; END_IF;
   "IEC_Timer_0_DB_50".TON(IN := ("SEQ_MAIN" = 9) AND NOT "OUTPUTS".LH_BOTTOM_CYL AND NOT "INPUTS".LH_BOTTOM_CYL_DOWN,
                           PT := T#2S);
   IF "IEC_Timer_0_DB_50".Q THEN "HMI INTERFACE".ERROR := 7; END_IF;
   "IEC_Timer_0_DB_49".TON(IN := ("SEQ_MAIN" = 13) AND NOT "OUTPUTS".LOCK3 AND NOT "INPUTS".LOCK3_REV,
                           PT := T#2S);
   IF "IEC_Timer_0_DB_49".Q THEN "HMI INTERFACE".ERROR := 5; END_IF;
   "IEC_Timer_0_DB_48".TON(IN := ("SEQ_MAIN" = 9) AND NOT "OUTPUTS".LOCK1 AND NOT "INPUTS".LOCK1_REV,
                           PT := T#2S);
   IF "IEC_Timer_0_DB_48".Q THEN "HMI INTERFACE".ERROR := 1; END_IF;
   #ERROR_BIT1 := "IEC_Timer_0_DB_42".Q OR "IEC_Timer_0_DB_43".Q OR "IEC_Timer_0_DB_44".Q OR "IEC_Timer_0_DB_47".Q OR "IEC_Timer_0_DB_46".Q OR "IEC_Timer_0_DB_45".Q OR "IEC_Timer_0_DB_51".Q OR "IEC_Timer_0_DB_50".Q OR "IEC_Timer_0_DB_49".Q OR "IEC_Timer_0_DB_48".Q;
END_REGION

REGION Network 2: ERROR_POPUP_ADDRESS
   RUNG wire#powerrail
      I_Contact( #ERROR_BIT1 )
      Coil( "HMI INTERFACE".ERROR_POPUP )
   END_RUNG
   // the same network as SCL:
   "HMI INTERFACE".ERROR_POPUP := NOT #ERROR_BIT1;
END_REGION
END_FUNCTION

FUNCTION "CVX 300 CAMERA" : Void   // FC5, LAD
{ S7_Optimized_Access := 'TRUE' }
VERSION : 0.1
   VAR_INPUT
      "CAM1 TRG" : Bool;
      "CAM2 TRG" : Bool;
      PROG_EN : Bool;
      PROG_NO : Int;
   END_VAR
   VAR_OUTPUT
      LOGO_RSLT_OK : Bool;
      LOGO_RSLT_NG : Bool;
      LED_RSLT_OK : Bool;
      LED_RSLT_NG : Bool;
   END_VAR
BEGIN

REGION Network 2: CAM_TRG
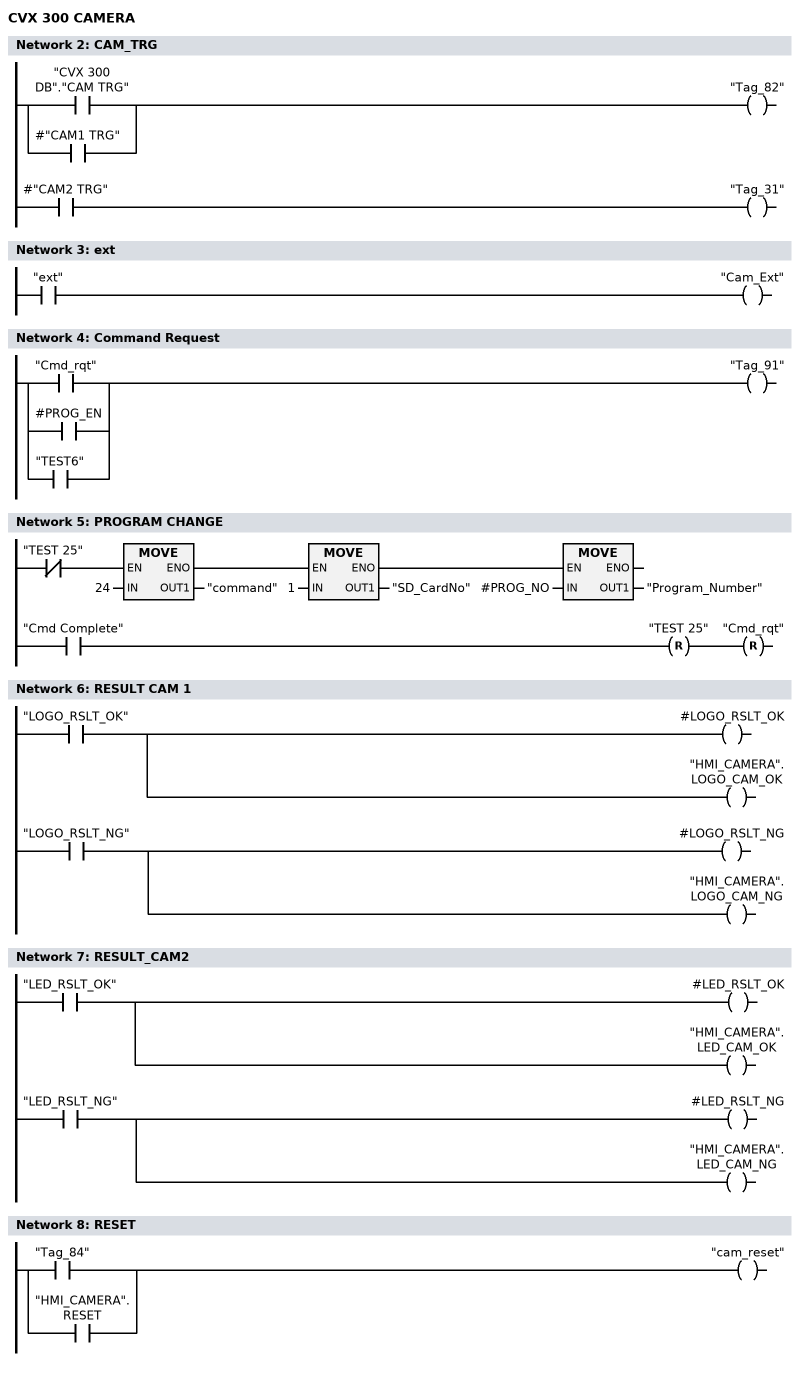
   RUNG wire#powerrail
      Contact( "CVX 300 DB"."CAM TRG" )
      wire#w1
      Coil( "Tag_82" )
   END_RUNG
   RUNG wire#powerrail
      Contact( #"CAM1 TRG" )
   END_RUNG wire#w1
   RUNG wire#powerrail
      Contact( #"CAM2 TRG" )
      Coil( "Tag_31" )
   END_RUNG
   // the same network as SCL:
   "Tag_82" := "CVX 300 DB"."CAM TRG" OR #"CAM1 TRG";
   "Tag_31" := #"CAM2 TRG";
END_REGION

REGION Network 3: ext
   RUNG wire#powerrail
      Contact( "ext" )
      Coil( "Cam_Ext" )
   END_RUNG
   // the same network as SCL:
   "Cam_Ext" := "ext";
END_REGION

REGION Network 4: Command Request
   RUNG wire#powerrail
      Contact( "Cmd_rqt" )
      wire#w1
      Coil( "Tag_91" )
   END_RUNG
   RUNG wire#powerrail
      Contact( #PROG_EN )
   END_RUNG wire#w1
   RUNG wire#powerrail
      Contact( "TEST6" )
   END_RUNG wire#w1
   // the same network as SCL:
   "Tag_91" := "Cmd_rqt" OR #PROG_EN OR "TEST6";
END_REGION

REGION Network 5: PROGRAM CHANGE
   RUNG wire#powerrail
      I_Contact( "TEST 25" )
      Move(in := 24, out1 => "command")
      Move(in := 1, out1 => "SD_CardNo")
      Move(in := #PROG_NO, out1 => "Program_Number")
   END_RUNG
   RUNG wire#powerrail
      Contact( "Cmd Complete" )
      R_Coil( "TEST 25" )
      R_Coil( "Cmd_rqt" )
   END_RUNG
   // the same network as SCL:
   IF NOT "TEST 25" THEN
       "command" := 24;
       "SD_CardNo" := 1;
       "Program_Number" := #PROG_NO;
   END_IF;
   IF "Cmd Complete" THEN
       "TEST 25" := FALSE;
       "Cmd_rqt" := FALSE;
   END_IF;
END_REGION

REGION Network 6: RESULT CAM 1
   RUNG wire#powerrail
      Contact( "LOGO_RSLT_OK" )
      wire#w1
      Coil( #LOGO_RSLT_OK )
   END_RUNG
   RUNG wire#w1
      Coil( "HMI_CAMERA".LOGO_CAM_OK )
   END_RUNG
   RUNG wire#powerrail
      Contact( "LOGO_RSLT_NG" )
      wire#w2
      Coil( #LOGO_RSLT_NG )
   END_RUNG
   RUNG wire#w2
      Coil( "HMI_CAMERA".LOGO_CAM_NG )
   END_RUNG
   // the same network as SCL:
   #LOGO_RSLT_OK := "LOGO_RSLT_OK";
   "HMI_CAMERA".LOGO_CAM_OK := "LOGO_RSLT_OK";
   #LOGO_RSLT_NG := "LOGO_RSLT_NG";
   "HMI_CAMERA".LOGO_CAM_NG := "LOGO_RSLT_NG";
END_REGION

REGION Network 7: RESULT_CAM2
   RUNG wire#powerrail
      Contact( "LED_RSLT_OK" )
      wire#w1
      Coil( #LED_RSLT_OK )
   END_RUNG
   RUNG wire#w1
      Coil( "HMI_CAMERA".LED_CAM_OK )
   END_RUNG
   RUNG wire#powerrail
      Contact( "LED_RSLT_NG" )
      wire#w2
      Coil( #LED_RSLT_NG )
   END_RUNG
   RUNG wire#w2
      Coil( "HMI_CAMERA".LED_CAM_NG )
   END_RUNG
   // the same network as SCL:
   #LED_RSLT_OK := "LED_RSLT_OK";
   "HMI_CAMERA".LED_CAM_OK := "LED_RSLT_OK";
   #LED_RSLT_NG := "LED_RSLT_NG";
   "HMI_CAMERA".LED_CAM_NG := "LED_RSLT_NG";
END_REGION

REGION Network 8: RESET
   RUNG wire#powerrail
      Contact( "Tag_84" )
      wire#w1
      Coil( "cam_reset" )
   END_RUNG
   RUNG wire#powerrail
      Contact( "HMI_CAMERA".RESET )
   END_RUNG wire#w1
   // the same network as SCL:
   "cam_reset" := "Tag_84" OR "HMI_CAMERA".RESET;
END_REGION
END_FUNCTION

ORGANIZATION_BLOCK "Main"   // OB1, LAD, ProgramCycle
TITLE = "Main Program Sweep (Cycle)"
{ S7_Optimized_Access := 'TRUE' }
VERSION : 0.1
   VAR_INPUT
      Initial_Call : Bool;   // Initial call of this OB
      Remanence : Bool;   // =True, if remanent data are available
   END_VAR
   VAR_TEMP
      ELE_CAL_RESET : Bool;
   END_VAR
   VAR_TEMP   // added for the SCL form of the ladder/FBD networks
      _w1 : Bool;
      _w2 : Bool;
      _w3 : Bool;
   END_VAR
BEGIN

REGION Network 2: TESTING SEQUENCE
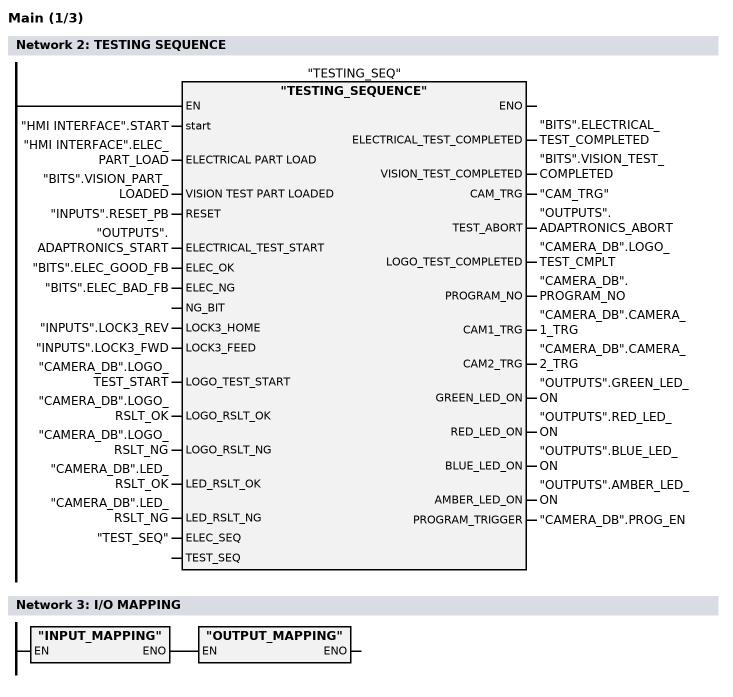
   RUNG wire#powerrail
      "TESTING_SEQ"(start := "HMI INTERFACE".START, "ELECTRICAL PART LOAD" := "HMI INTERFACE".ELEC_PART_LOAD, "VISION TEST PART LOADED" := "BITS".VISION_PART_LOADED, RESET := "INPUTS".RESET_PB, ELECTRICAL_TEST_START := "OUTPUTS".ADAPTRONICS_START, ELEC_OK := "BITS".ELEC_GOOD_FB, ELEC_NG := "BITS".ELEC_BAD_FB, NG_BIT :=, LOCK3_HOME := "INPUTS".LOCK3_REV, LOCK3_FEED := "INPUTS".LOCK3_FWD, LOGO_TEST_START := "CAMERA_DB".LOGO_TEST_START, LOGO_RSLT_OK := "CAMERA_DB".LOGO_RSLT_OK, LOGO_RSLT_NG := "CAMERA_DB".LOGO_RSLT_NG, LED_RSLT_OK := "CAMERA_DB".LED_RSLT_OK, LED_RSLT_NG := "CAMERA_DB".LED_RSLT_NG, ELEC_SEQ := "TEST_SEQ", TEST_SEQ :=, ELECTRICAL_TEST_COMPLETED => "BITS".ELECTRICAL_TEST_COMPLETED, VISION_TEST_COMPLETED => "BITS".VISION_TEST_COMPLETED, CAM_TRG => "CAM_TRG", TEST_ABORT => "OUTPUTS".ADAPTRONICS_ABORT, LOGO_TEST_COMPLETED => "CAMERA_DB".LOGO_TEST_CMPLT, PROGRAM_NO => "CAMERA_DB".PROGRAM_NO, CAM1_TRG => "CAMERA_DB".CAMERA_1_TRG, CAM2_TRG => "CAMERA_DB".CAMERA_2_TRG, GREEN_LED_ON => "OUTPUTS".GREEN_LED_ON, RED_LED_ON => "OUTPUTS".RED_LED_ON, BLUE_LED_ON => "OUTPUTS".BLUE_LED_ON, AMBER_LED_ON => "OUTPUTS".AMBER_LED_ON, PROGRAM_TRIGGER => "CAMERA_DB".PROG_EN)
   END_RUNG
   // the same network as SCL:
   "TESTING_SEQ"(start := "HMI INTERFACE".START,   // "TESTING_SEQUENCE"
                 "ELECTRICAL PART LOAD" := "HMI INTERFACE".ELEC_PART_LOAD,
                 "VISION TEST PART LOADED" := "BITS".VISION_PART_LOADED,
                 RESET := "INPUTS".RESET_PB,
                 ELECTRICAL_TEST_START := "OUTPUTS".ADAPTRONICS_START,
                 ELEC_OK := "BITS".ELEC_GOOD_FB,
                 ELEC_NG := "BITS".ELEC_BAD_FB,
                 LOCK3_HOME := "INPUTS".LOCK3_REV,
                 LOCK3_FEED := "INPUTS".LOCK3_FWD,
                 LOGO_TEST_START := "CAMERA_DB".LOGO_TEST_START,
                 LOGO_RSLT_OK := "CAMERA_DB".LOGO_RSLT_OK,
                 LOGO_RSLT_NG := "CAMERA_DB".LOGO_RSLT_NG,
                 LED_RSLT_OK := "CAMERA_DB".LED_RSLT_OK,
                 LED_RSLT_NG := "CAMERA_DB".LED_RSLT_NG,
                 ELEC_SEQ := "TEST_SEQ",
                 ELECTRICAL_TEST_COMPLETED => "BITS".ELECTRICAL_TEST_COMPLETED,
                 VISION_TEST_COMPLETED => "BITS".VISION_TEST_COMPLETED,
                 CAM_TRG => "CAM_TRG",
                 TEST_ABORT => "OUTPUTS".ADAPTRONICS_ABORT,
                 LOGO_TEST_COMPLETED => "CAMERA_DB".LOGO_TEST_CMPLT,
                 PROGRAM_NO => "CAMERA_DB".PROGRAM_NO,
                 CAM1_TRG => "CAMERA_DB".CAMERA_1_TRG,
                 CAM2_TRG => "CAMERA_DB".CAMERA_2_TRG,
                 GREEN_LED_ON => "OUTPUTS".GREEN_LED_ON,
                 RED_LED_ON => "OUTPUTS".RED_LED_ON,
                 BLUE_LED_ON => "OUTPUTS".BLUE_LED_ON,
                 AMBER_LED_ON => "OUTPUTS".AMBER_LED_ON,
                 PROGRAM_TRIGGER => "CAMERA_DB".PROG_EN);
END_REGION

REGION Network 3: I/O MAPPING
   RUNG wire#powerrail
      "INPUT_MAPPING"()
      "OUTPUT_MAPPING"()
   END_RUNG
   // the same network as SCL:
   "INPUT_MAPPING"(ENO => #_w1);
   IF #_w1 THEN "OUTPUT_MAPPING"(); END_IF;
END_REGION

REGION Network 4: MAIN_SEQUENCE
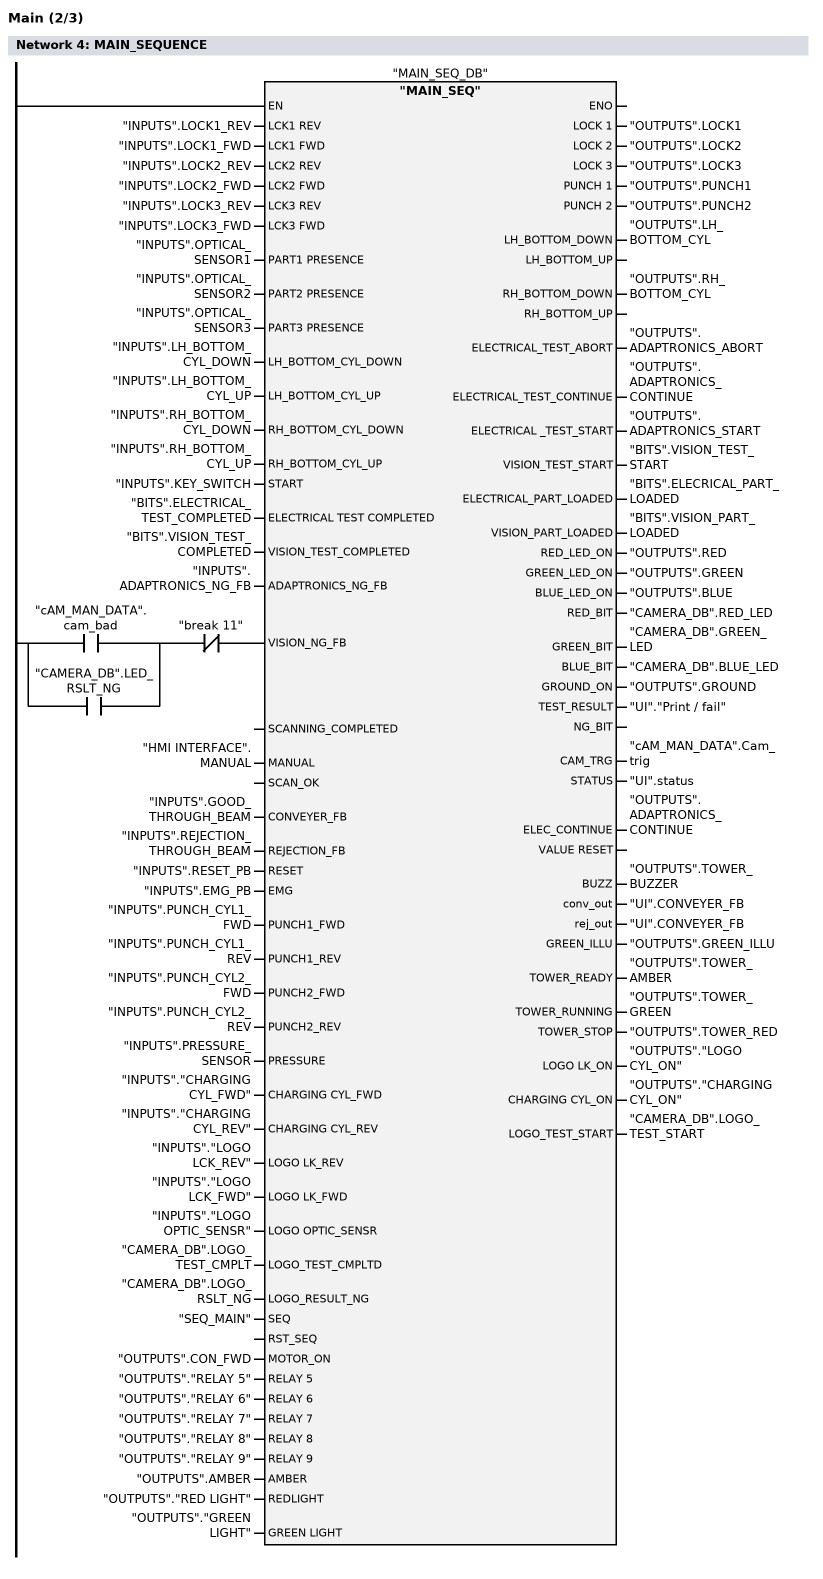
   RUNG wire#powerrail
      "MAIN_SEQ_DB"(VISION_NG_FB := wire#w2, "LCK1 REV" := "INPUTS".LOCK1_REV, "LCK1 FWD" := "INPUTS".LOCK1_FWD, "LCK2 REV" := "INPUTS".LOCK2_REV, "LCK2 FWD" := "INPUTS".LOCK2_FWD, "LCK3 REV" := "INPUTS".LOCK3_REV, "LCK3 FWD" := "INPUTS".LOCK3_FWD, "PART1 PRESENCE" := "INPUTS".OPTICAL_SENSOR1, "PART2 PRESENCE" := "INPUTS".OPTICAL_SENSOR2, "PART3 PRESENCE" := "INPUTS".OPTICAL_SENSOR3, LH_BOTTOM_CYL_DOWN := "INPUTS".LH_BOTTOM_CYL_DOWN, LH_BOTTOM_CYL_UP := "INPUTS".LH_BOTTOM_CYL_UP, RH_BOTTOM_CYL_DOWN := "INPUTS".RH_BOTTOM_CYL_DOWN, RH_BOTTOM_CYL_UP := "INPUTS".RH_BOTTOM_CYL_UP, START := "INPUTS".KEY_SWITCH, "ELECTRICAL TEST COMPLETED" := "BITS".ELECTRICAL_TEST_COMPLETED, VISION_TEST_COMPLETED := "BITS".VISION_TEST_COMPLETED, ADAPTRONICS_NG_FB := "INPUTS".ADAPTRONICS_NG_FB, SCANNING_COMPLETED :=, MANUAL := "HMI INTERFACE".MANUAL, SCAN_OK :=, CONVEYER_FB := "INPUTS".GOOD_THROUGH_BEAM, REJECTION_FB := "INPUTS".REJECTION_THROUGH_BEAM, RESET := "INPUTS".RESET_PB, EMG := "INPUTS".EMG_PB, PUNCH1_FWD := "INPUTS".PUNCH_CYL1_FWD, PUNCH1_REV := "INPUTS".PUNCH_CYL1_REV, PUNCH2_FWD := "INPUTS".PUNCH_CYL2_FWD, PUNCH2_REV := "INPUTS".PUNCH_CYL2_REV, PRESSURE := "INPUTS".PRESSURE_SENSOR, "CHARGING CYL_FWD" := "INPUTS"."CHARGING CYL_FWD", "CHARGING CYL_REV" := "INPUTS"."CHARGING CYL_REV", "LOGO LK_REV" := "INPUTS"."LOGO LCK_REV", "LOGO LK_FWD" := "INPUTS"."LOGO LCK_FWD", "LOGO OPTIC_SENSR" := "INPUTS"."LOGO OPTIC_SENSR", LOGO_TEST_CMPLTD := "CAMERA_DB".LOGO_TEST_CMPLT, LOGO_RESULT_NG := "CAMERA_DB".LOGO_RSLT_NG, SEQ := "SEQ_MAIN", RST_SEQ :=, MOTOR_ON := "OUTPUTS".CON_FWD, "RELAY 5" := "OUTPUTS"."RELAY 5", "RELAY 6" := "OUTPUTS"."RELAY 6", "RELAY 7" := "OUTPUTS"."RELAY 7", "RELAY 8" := "OUTPUTS"."RELAY 8", "RELAY 9" := "OUTPUTS"."RELAY 9", AMBER := "OUTPUTS".AMBER, REDLIGHT := "OUTPUTS"."RED LIGHT", "GREEN LIGHT" := "OUTPUTS"."GREEN LIGHT", "LOCK 1" => "OUTPUTS".LOCK1, "LOCK 2" => "OUTPUTS".LOCK2, "LOCK 3" => "OUTPUTS".LOCK3, "PUNCH 1" => "OUTPUTS".PUNCH1, "PUNCH 2" => "OUTPUTS".PUNCH2, LH_BOTTOM_DOWN => "OUTPUTS".LH_BOTTOM_CYL, LH_BOTTOM_UP =>, RH_BOTTOM_DOWN => "OUTPUTS".RH_BOTTOM_CYL, RH_BOTTOM_UP =>, ELECTRICAL_TEST_ABORT => "OUTPUTS".ADAPTRONICS_ABORT, ELECTRICAL_TEST_CONTINUE => "OUTPUTS".ADAPTRONICS_CONTINUE, "ELECTRICAL _TEST_START" => "OUTPUTS".ADAPTRONICS_START, VISION_TEST_START => "BITS".VISION_TEST_START, ELECTRICAL_PART_LOADED => "BITS".ELECRICAL_PART_LOADED, VISION_PART_LOADED => "BITS".VISION_PART_LOADED, RED_LED_ON => "OUTPUTS".RED, GREEN_LED_ON => "OUTPUTS".GREEN, BLUE_LED_ON => "OUTPUTS".BLUE, RED_BIT => "CAMERA_DB".RED_LED, GREEN_BIT => "CAMERA_DB".GREEN_LED, BLUE_BIT => "CAMERA_DB".BLUE_LED, GROUND_ON => "OUTPUTS".GROUND, TEST_RESULT => "UI"."Print / fail", NG_BIT =>, CAM_TRG => "cAM_MAN_DATA".Cam_trig, STATUS => "UI".status, ELEC_CONTINUE => "OUTPUTS".ADAPTRONICS_CONTINUE, "VALUE RESET" =>, BUZZ => "OUTPUTS".TOWER_BUZZER, conv_out => "UI".CONVEYER_FB, rej_out => "UI".CONVEYER_FB, GREEN_ILLU => "OUTPUTS".GREEN_ILLU, TOWER_READY => "OUTPUTS".TOWER_AMBER, TOWER_RUNNING => "OUTPUTS".TOWER_GREEN, TOWER_STOP => "OUTPUTS".TOWER_RED, "LOGO LK_ON" => "OUTPUTS"."LOGO CYL_ON", "CHARGING CYL_ON" => "OUTPUTS"."CHARGING CYL_ON", LOGO_TEST_START => "CAMERA_DB".LOGO_TEST_START)
   END_RUNG
   RUNG wire#powerrail
      Contact( "cAM_MAN_DATA".cam_bad )
      wire#w1
      I_Contact( "break 11" )
   END_RUNG wire#w2
   RUNG wire#powerrail
      Contact( "CAMERA_DB".LED_RSLT_NG )
   END_RUNG wire#w1
   // the same network as SCL:
   "MAIN_SEQ_DB"("LCK1 REV" := "INPUTS".LOCK1_REV,   // "MAIN_SEQ"
                 "LCK1 FWD" := "INPUTS".LOCK1_FWD,
                 "LCK2 REV" := "INPUTS".LOCK2_REV,
                 "LCK2 FWD" := "INPUTS".LOCK2_FWD,
                 "LCK3 REV" := "INPUTS".LOCK3_REV,
                 "LCK3 FWD" := "INPUTS".LOCK3_FWD,
                 "PART1 PRESENCE" := "INPUTS".OPTICAL_SENSOR1,
                 "PART2 PRESENCE" := "INPUTS".OPTICAL_SENSOR2,
                 "PART3 PRESENCE" := "INPUTS".OPTICAL_SENSOR3,
                 LH_BOTTOM_CYL_DOWN := "INPUTS".LH_BOTTOM_CYL_DOWN,
                 LH_BOTTOM_CYL_UP := "INPUTS".LH_BOTTOM_CYL_UP,
                 RH_BOTTOM_CYL_DOWN := "INPUTS".RH_BOTTOM_CYL_DOWN,
                 RH_BOTTOM_CYL_UP := "INPUTS".RH_BOTTOM_CYL_UP,
                 START := "INPUTS".KEY_SWITCH,
                 "ELECTRICAL TEST COMPLETED" := "BITS".ELECTRICAL_TEST_COMPLETED,
                 VISION_TEST_COMPLETED := "BITS".VISION_TEST_COMPLETED,
                 ADAPTRONICS_NG_FB := "INPUTS".ADAPTRONICS_NG_FB,
                 VISION_NG_FB := ("cAM_MAN_DATA".cam_bad OR "CAMERA_DB".LED_RSLT_NG) AND NOT "break 11",
                 MANUAL := "HMI INTERFACE".MANUAL,
                 CONVEYER_FB := "INPUTS".GOOD_THROUGH_BEAM,
                 REJECTION_FB := "INPUTS".REJECTION_THROUGH_BEAM,
                 RESET := "INPUTS".RESET_PB,
                 EMG := "INPUTS".EMG_PB,
                 PUNCH1_FWD := "INPUTS".PUNCH_CYL1_FWD,
                 PUNCH1_REV := "INPUTS".PUNCH_CYL1_REV,
                 PUNCH2_FWD := "INPUTS".PUNCH_CYL2_FWD,
                 PUNCH2_REV := "INPUTS".PUNCH_CYL2_REV,
                 PRESSURE := "INPUTS".PRESSURE_SENSOR,
                 "CHARGING CYL_FWD" := "INPUTS"."CHARGING CYL_FWD",
                 "CHARGING CYL_REV" := "INPUTS"."CHARGING CYL_REV",
                 "LOGO LK_REV" := "INPUTS"."LOGO LCK_REV",
                 "LOGO LK_FWD" := "INPUTS"."LOGO LCK_FWD",
                 "LOGO OPTIC_SENSR" := "INPUTS"."LOGO OPTIC_SENSR",
                 LOGO_TEST_CMPLTD := "CAMERA_DB".LOGO_TEST_CMPLT,
                 LOGO_RESULT_NG := "CAMERA_DB".LOGO_RSLT_NG,
                 SEQ := "SEQ_MAIN",
                 MOTOR_ON := "OUTPUTS".CON_FWD,
                 "RELAY 5" := "OUTPUTS"."RELAY 5",
                 "RELAY 6" := "OUTPUTS"."RELAY 6",
                 "RELAY 7" := "OUTPUTS"."RELAY 7",
                 "RELAY 8" := "OUTPUTS"."RELAY 8",
                 "RELAY 9" := "OUTPUTS"."RELAY 9",
                 AMBER := "OUTPUTS".AMBER,
                 REDLIGHT := "OUTPUTS"."RED LIGHT",
                 "GREEN LIGHT" := "OUTPUTS"."GREEN LIGHT",
                 "LOCK 1" => "OUTPUTS".LOCK1,
                 "LOCK 2" => "OUTPUTS".LOCK2,
                 "LOCK 3" => "OUTPUTS".LOCK3,
                 "PUNCH 1" => "OUTPUTS".PUNCH1,
                 "PUNCH 2" => "OUTPUTS".PUNCH2,
                 LH_BOTTOM_DOWN => "OUTPUTS".LH_BOTTOM_CYL,
                 RH_BOTTOM_DOWN => "OUTPUTS".RH_BOTTOM_CYL,
                 ELECTRICAL_TEST_ABORT => "OUTPUTS".ADAPTRONICS_ABORT,
                 ELECTRICAL_TEST_CONTINUE => "OUTPUTS".ADAPTRONICS_CONTINUE,
                 "ELECTRICAL _TEST_START" => "OUTPUTS".ADAPTRONICS_START,
                 VISION_TEST_START => "BITS".VISION_TEST_START,
                 ELECTRICAL_PART_LOADED => "BITS".ELECRICAL_PART_LOADED,
                 VISION_PART_LOADED => "BITS".VISION_PART_LOADED,
                 RED_LED_ON => "OUTPUTS".RED,
                 GREEN_LED_ON => "OUTPUTS".GREEN,
                 BLUE_LED_ON => "OUTPUTS".BLUE,
                 RED_BIT => "CAMERA_DB".RED_LED,
                 GREEN_BIT => "CAMERA_DB".GREEN_LED,
                 BLUE_BIT => "CAMERA_DB".BLUE_LED,
                 GROUND_ON => "OUTPUTS".GROUND,
                 TEST_RESULT => "UI"."Print / fail",
                 CAM_TRG => "cAM_MAN_DATA".Cam_trig,
                 STATUS => "UI".status,
                 ELEC_CONTINUE => "OUTPUTS".ADAPTRONICS_CONTINUE,
                 BUZZ => "OUTPUTS".TOWER_BUZZER,
                 conv_out => "UI".CONVEYER_FB,
                 rej_out => "UI".CONVEYER_FB,
                 GREEN_ILLU => "OUTPUTS".GREEN_ILLU,
                 TOWER_READY => "OUTPUTS".TOWER_AMBER,
                 TOWER_RUNNING => "OUTPUTS".TOWER_GREEN,
                 TOWER_STOP => "OUTPUTS".TOWER_RED,
                 "LOGO LK_ON" => "OUTPUTS"."LOGO CYL_ON",
                 "CHARGING CYL_ON" => "OUTPUTS"."CHARGING CYL_ON",
                 LOGO_TEST_START => "CAMERA_DB".LOGO_TEST_START);
END_REGION

REGION Network 5: ERROR_MESSAGES
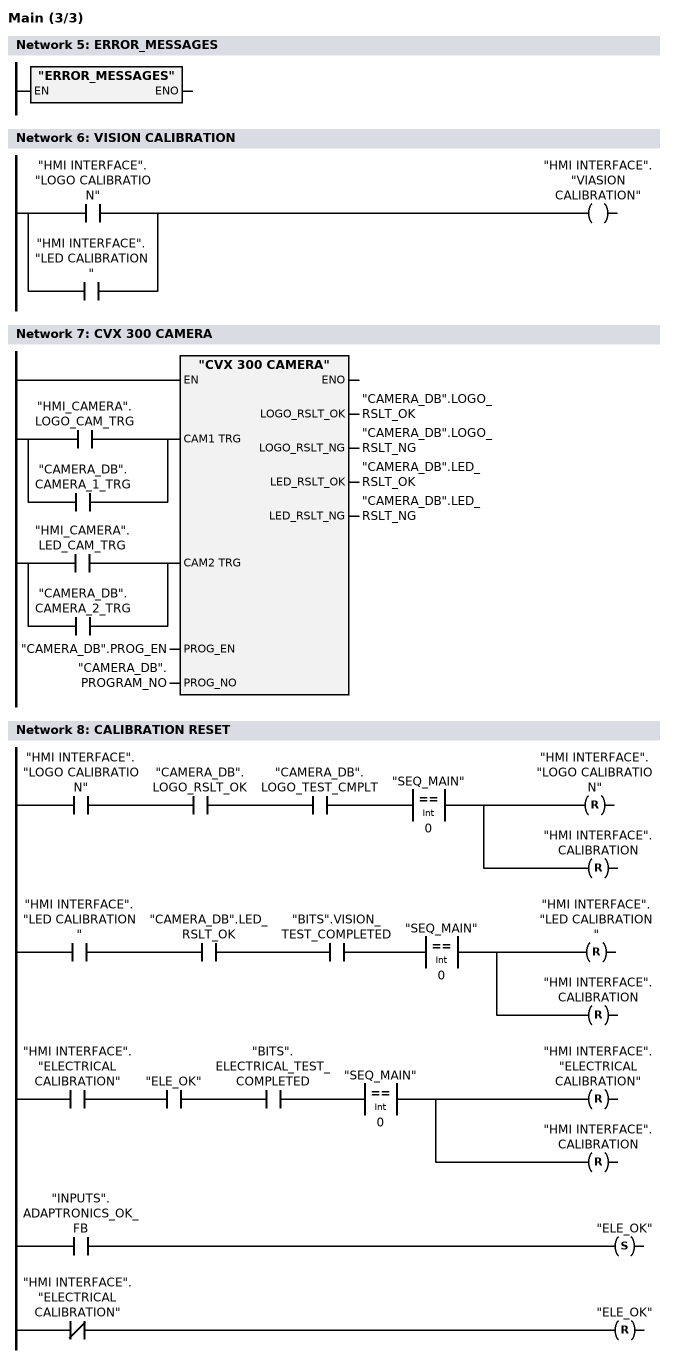
   RUNG wire#powerrail
      "ERROR_MESSAGES"()
   END_RUNG
   // the same network as SCL:
   "ERROR_MESSAGES"();
END_REGION

REGION Network 6: VISION CALIBRATION
   RUNG wire#powerrail
      Contact( "HMI INTERFACE"."LOGO CALIBRATION" )
      wire#w1
      Coil( "HMI INTERFACE"."VIASION CALIBRATION" )
   END_RUNG
   RUNG wire#powerrail
      Contact( "HMI INTERFACE"."LED CALIBRATION" )
   END_RUNG wire#w1
   // the same network as SCL:
   "HMI INTERFACE"."VIASION CALIBRATION" := "HMI INTERFACE"."LOGO CALIBRATION" OR "HMI INTERFACE"."LED CALIBRATION";
END_REGION

REGION Network 7: CVX 300 CAMERA
   RUNG wire#powerrail
      "CVX 300 CAMERA"("CAM1 TRG" := wire#w1, "CAM2 TRG" := wire#w2, PROG_EN := "CAMERA_DB".PROG_EN, PROG_NO := "CAMERA_DB".PROGRAM_NO, LOGO_RSLT_OK => "CAMERA_DB".LOGO_RSLT_OK, LOGO_RSLT_NG => "CAMERA_DB".LOGO_RSLT_NG, LED_RSLT_OK => "CAMERA_DB".LED_RSLT_OK, LED_RSLT_NG => "CAMERA_DB".LED_RSLT_NG)
   END_RUNG
   RUNG wire#powerrail
      Contact( "HMI_CAMERA".LOGO_CAM_TRG )
   END_RUNG wire#w1
   RUNG wire#powerrail
      Contact( "CAMERA_DB".CAMERA_1_TRG )
   END_RUNG wire#w1
   RUNG wire#powerrail
      Contact( "HMI_CAMERA".LED_CAM_TRG )
   END_RUNG wire#w2
   RUNG wire#powerrail
      Contact( "CAMERA_DB".CAMERA_2_TRG )
   END_RUNG wire#w2
   // the same network as SCL:
   "CVX 300 CAMERA"("CAM1 TRG" := "HMI_CAMERA".LOGO_CAM_TRG OR "CAMERA_DB".CAMERA_1_TRG,
                    "CAM2 TRG" := "HMI_CAMERA".LED_CAM_TRG OR "CAMERA_DB".CAMERA_2_TRG,
                    PROG_EN := "CAMERA_DB".PROG_EN,
                    PROG_NO := "CAMERA_DB".PROGRAM_NO,
                    LOGO_RSLT_OK => "CAMERA_DB".LOGO_RSLT_OK,
                    LOGO_RSLT_NG => "CAMERA_DB".LOGO_RSLT_NG,
                    LED_RSLT_OK => "CAMERA_DB".LED_RSLT_OK,
                    LED_RSLT_NG => "CAMERA_DB".LED_RSLT_NG);
END_REGION

REGION Network 8: CALIBRATION RESET
   RUNG wire#powerrail
      Contact( "HMI INTERFACE"."LOGO CALIBRATION" )
      Contact( "CAMERA_DB".LOGO_RSLT_OK )
      Contact( "CAMERA_DB".LOGO_TEST_CMPLT )
      { S7_Templates := "SrcType := Int" } EQ_Contact(in1 := "SEQ_MAIN", in2 := 0)
      wire#w1
      R_Coil( "HMI INTERFACE"."LOGO CALIBRATION" )
   END_RUNG
   RUNG wire#w1
      R_Coil( "HMI INTERFACE".CALIBRATION )
   END_RUNG
   RUNG wire#powerrail
      Contact( "HMI INTERFACE"."LED CALIBRATION" )
      Contact( "CAMERA_DB".LED_RSLT_OK )
      Contact( "BITS".VISION_TEST_COMPLETED )
      { S7_Templates := "SrcType := Int" } EQ_Contact(in1 := "SEQ_MAIN", in2 := 0)
      wire#w2
      R_Coil( "HMI INTERFACE"."LED CALIBRATION" )
   END_RUNG
   RUNG wire#w2
      R_Coil( "HMI INTERFACE".CALIBRATION )
   END_RUNG
   RUNG wire#powerrail
      Contact( "HMI INTERFACE"."ELECTRICAL CALIBRATION" )
      Contact( "ELE_OK" )
      Contact( "BITS".ELECTRICAL_TEST_COMPLETED )
      { S7_Templates := "SrcType := Int" } EQ_Contact(in1 := "SEQ_MAIN", in2 := 0)
      wire#w3
      R_Coil( "HMI INTERFACE"."ELECTRICAL CALIBRATION" )
   END_RUNG
   RUNG wire#w3
      R_Coil( "HMI INTERFACE".CALIBRATION )
   END_RUNG
   RUNG wire#powerrail
      Contact( "INPUTS".ADAPTRONICS_OK_FB )
      S_Coil( "ELE_OK" )
   END_RUNG
   RUNG wire#powerrail
      I_Contact( "HMI INTERFACE"."ELECTRICAL CALIBRATION" )
      R_Coil( "ELE_OK" )
   END_RUNG
   // the same network as SCL:
   #_w1 := "HMI INTERFACE"."LOGO CALIBRATION" AND "CAMERA_DB".LOGO_RSLT_OK AND "CAMERA_DB".LOGO_TEST_CMPLT AND ("SEQ_MAIN" = 0);
   IF #_w1 THEN
       "HMI INTERFACE"."LOGO CALIBRATION" := FALSE;
       "HMI INTERFACE".CALIBRATION := FALSE;
   END_IF;
   #_w2 := "HMI INTERFACE"."LED CALIBRATION" AND "CAMERA_DB".LED_RSLT_OK AND "BITS".VISION_TEST_COMPLETED AND ("SEQ_MAIN" = 0);
   IF #_w2 THEN
       "HMI INTERFACE"."LED CALIBRATION" := FALSE;
       "HMI INTERFACE".CALIBRATION := FALSE;
   END_IF;
   #_w3 := "HMI INTERFACE"."ELECTRICAL CALIBRATION" AND "ELE_OK" AND "BITS".ELECTRICAL_TEST_COMPLETED AND ("SEQ_MAIN" = 0);
   IF #_w3 THEN
       "HMI INTERFACE"."ELECTRICAL CALIBRATION" := FALSE;
       "HMI INTERFACE".CALIBRATION := FALSE;
   END_IF;
   IF "INPUTS".ADAPTRONICS_OK_FB THEN "ELE_OK" := TRUE; END_IF;
   IF NOT "HMI INTERFACE"."ELECTRICAL CALIBRATION" THEN "ELE_OK" := FALSE; END_IF;
END_REGION
END_ORGANIZATION_BLOCK